LIN {X 0,Y 277.83,Z 467.311,A -85,B 0,C 180,E1 -25540.628,E2 -25540.628} C_VEL
LIN {X 0,Y 277.38,Z 485.512,A -85,B 0,C 180,E1 -25541.504,E2 -25541.504} C_VEL
LIN {X 0,Y 276.723,Z 501.553,A -85,B 0,C 180,E1 -25542.602,E2 -25542.602} C_VEL
LIN {X 0,Y 276.071,Z 515.024,A -85,B 0,C 180,E1 -25543.794,E2 -25543.794} C_VEL
LIN {X 0,Y 275.265,Z 529.451,A -85,B 0,C 180,E1 -25545.393,E2 -25545.393} C_VEL
LIN {X 0,Y 274.573,Z 543.321,A -85,B 0,C 180,E1 -25547.289,E2 -25547.289} C_VEL
LIN {X 0,Y 273.841,Z 555.486,A -85,B 0,C 180,E1 -25549.313,E2 -25549.313} C_VEL
LIN {X 0,Y 273.731,Z 556.96,A -85,B 0,C 180,E1 -25549.589,E2 -25549.589} C_VEL
LIN {X 0,Y 272.791,Z 561.229,A -85,B 0,C 180,E1 -25550.426,E2 -25550.426} C_VEL
LIN {X 0,Y 269.621,Z 567.675,A -85,B 0,C 180,E1 -25551.869,E2 -25551.869} C_VEL
LIN {X 0,Y 266.574,Z 573.805,A -85,B 0,C 180,E1 -25553.418,E2 -25553.418} C_VEL
LIN {X 0,Y 265.838,Z 577.453,A -85,B 0,C 180,E1 -25554.406,E2 -25554.406} C_VEL
LIN {X 0,Y 265.849,Z 586.101,A -85,B 0,C 180,E1 -25556.979,E2 -25556.979} C_VEL
LIN {X 0,Y 266.003,Z 592.424,A -85,B 0,C 180,E1 -25559.245,E2 -25559.245} C_VEL
LIN {X 0,Y 266.684,Z 599.311,A -85,B 0,C 180,E1 -25562.258,E2 -25562.258} C_VEL
LIN {X 0,Y 268.062,Z 604.601,A -85,B 0,C 180,E1 -25565.247,E2 -25565.247} C_VEL
LIN {X 0,Y 269.492,Z 607.656,A -85,B 0,C 180,E1 -25567.467,E2 -25567.467} C_VEL
LIN {X 0,Y 271.89,Z 610.479,A -85,B 0,C 180,E1 -25570.389,E2 -25570.389} C_VEL
LIN {X 0,Y 275.047,Z 611.982,A -85,B 0,C 180,E1 -25573.249,E2 -25573.249} C_VEL
LIN {X 0,Y 276.98,Z 612.223,A -85,B 0,C 180,E1 -25574.648,E2 -25574.648} C_VEL
LIN {X 0,Y 281.552,Z 611.672,A -85,B 0,C 180,E1 -25577.369,E2 -25577.369} C_VEL
LIN {X 0,Y 286.526,Z 609.815,A -85,B 0,C 180,E1 -25580.013,E2 -25580.013} C_VEL
LIN {X 0,Y 292.033,Z 606.641,A -85,B 0,C 180,E1 -25582.567,E2 -25582.567} C_VEL
LIN {X 0,Y 298.202,Z 601.947,A -85,B 0,C 180,E1 -25585.011,E2 -25585.011} C_VEL
LIN {X 0,Y 304.831,Z 595.719,A -85,B 0,C 180,E1 -25587.359,E2 -25587.359} C_VEL
LIN {X 0,Y 310.995,Z 588.827,A -85,B 0,C 180,E1 -25589.332,E2 -25589.332} C_VEL
LIN {X 0,Y 317.678,Z 580.405,A -85,B 0,C 180,E1 -25591.208,E2 -25591.208} C_VEL
LIN {X 0,Y 323.654,Z 571.647,A -85,B 0,C 180,E1 -25592.755,E2 -25592.755} C_VEL
LIN {X 0,Y 329.828,Z 561.351,A -85,B 0,C 180,E1 -25594.247,E2 -25594.247} C_VEL
LIN {X 0,Y 335.133,Z 551.118,A -85,B 0,C 180,E1 -25595.449,E2 -25595.449} C_VEL
LIN {X 0,Y 341.022,Z 537.921,A -85,B 0,C 180,E1 -25596.742,E2 -25596.742} C_VEL
LIN {X 0,Y 345.906,Z 524.621,A -85,B 0,C 180,E1 -25597.774,E2 -25597.774} C_VEL
LIN {X 0,Y 350.516,Z 508.978,A -85,B 0,C 180,E1 -25598.735,E2 -25598.735} C_VEL
LIN {X 0,Y 355.504,Z 486.941,A -85,B 0,C 180,E1 -25599.714,E2 -25599.714} C_VEL
LIN {X 0,Y 359.013,Z 471.3,A -85,B 0,C 180,E1 -25600.286,E2 -25600.286} C_VEL
LIN {X 0,Y 358.746,Z 470.474,A -85,B 0,C 180,E1 -25601.016,E2 -25601.016} C_VEL
LIN {X 0,Y 358.206,Z 469.756,A -85,B 0,C 180,E1 -25603.188,E2 -25603.188} C_VEL
LIN {X 0,Y 358.394,Z 470.084,A -85,B 0,C 180,E1 -25604.963,E2 -25604.963} C_VEL
LIN {X 0,Y 358.539,Z 470.42,A -85,B 0,C 180,E1 -25605.572,E2 -25605.572} C_VEL
LIN {X 0,Y 355.174,Z 487.615,A -85,B 0,C 180,E1 -25607.063,E2 -25607.063} C_VEL
LIN {X 0,Y 352.734,Z 500.618,A -85,B 0,C 180,E1 -25607.993,E2 -25607.993} C_VEL
LIN {X 0,Y 351.508,Z 506.79,A -85,B 0,C 180,E1 -25608.315,E2 -25608.315} C_VEL
LIN {X 0,Y 346.503,Z 527.149,A -85,B 0,C 180,E1 -25609.055,E2 -25609.055} C_VEL
LIN {X 0,Y 340.345,Z 545.929,A -85,B 0,C 180,E1 -25609.897,E2 -25609.897} C_VEL
LIN {X 0,Y 333.914,Z 561.533,A -85,B 0,C 180,E1 -25610.781,E2 -25610.781} C_VEL
LIN {X 0,Y 326.496,Z 576.813,A -85,B 0,C 180,E1 -25611.918,E2 -25611.918} C_VEL
LIN {X 0,Y 319.543,Z 589.349,A -85,B 0,C 180,E1 -25613.125,E2 -25613.125} C_VEL
LIN {X 0,Y 312.972,Z 599.943,A -85,B 0,C 180,E1 -25614.416,E2 -25614.416} C_VEL
LIN {X 0,Y 306.212,Z 609.968,A -85,B 0,C 180,E1 -25615.914,E2 -25615.914} C_VEL
LIN {X 0,Y 298.907,Z 619.806,A -85,B 0,C 180,E1 -25617.784,E2 -25617.784} C_VEL
LIN {X 0,Y 292.343,Z 628.114,A -85,B 0,C 180,E1 -25619.791,E2 -25619.791} C_VEL
LIN {X 0,Y 285.597,Z 635.955,A -85,B 0,C 180,E1 -25622.226,E2 -25622.226} C_VEL
LIN {X 0,Y 279.804,Z 642.289,A -85,B 0,C 180,E1 -25624.813,E2 -25624.813} C_VEL
LIN {X 0,Y 274.862,Z 647.227,A -85,B 0,C 180,E1 -25627.526,E2 -25627.526} C_VEL
LIN {X 0,Y 270.975,Z 650.909,A -85,B 0,C 180,E1 -25630.364,E2 -25630.364} C_VEL
LIN {X 0,Y 268.293,Z 653.413,A -85,B 0,C 180,E1 -25633.31,E2 -25633.31} C_VEL
LIN {X 0,Y 266.458,Z 654.808,A -85,B 0,C 180,E1 -25636.563,E2 -25636.563} C_VEL
LIN {X 0,Y 266.255,Z 655.027,A -85,B 0,C 180,E1 -25637.015,E2 -25637.015} C_VEL
LIN {X 0,Y 265.734,Z 658.417,A -85,B 0,C 180,E1 -25639.367,E2 -25639.367} C_VEL
LIN {X 0,Y 265.875,Z 660.76,A -85,B 0,C 180,E1 -25641.382,E2 -25641.382} C_VEL
LIN {X 0,Y 265.538,Z 670.158,A -85,B 0,C 180,E1 -25643.563,E2 -25643.563} C_VEL
LIN {X 0,Y 265.443,Z 678.349,A -85,B 0,C 180,E1 -25645.838,E2 -25645.838} C_VEL
LIN {X 0,Y 265.218,Z 686.104,A -85,B 0,C 180,E1 -25648.486,E2 -25648.486} C_VEL
LIN {X 0,Y 265.047,Z 691.433,A -85,B 0,C 180,E1 -25650.757,E2 -25650.757} C_VEL
LIN {X 0,Y 264.821,Z 696.988,A -85,B 0,C 180,E1 -25653.791,E2 -25653.791} C_VEL
LIN {X 0,Y 264.9,Z 700.153,A -85,B 0,C 180,E1 -25656.071,E2 -25656.071} C_VEL
LIN {X 0,Y 265.517,Z 703.155,A -85,B 0,C 180,E1 -25659.107,E2 -25659.107} C_VEL
LIN {X 0,Y 267.125,Z 704.904,A -85,B 0,C 180,E1 -25662.109,E2 -25662.109} C_VEL
LIN {X 0,Y 269.559,Z 705.406,A -85,B 0,C 180,E1 -25665.061,E2 -25665.061} C_VEL
LIN {X 0,Y 272.975,Z 704.659,A -85,B 0,C 180,E1 -25667.934,E2 -25667.934} C_VEL
LIN {X 0,Y 276.889,Z 702.698,A -85,B 0,C 180,E1 -25670.742,E2 -25670.742} C_VEL
LIN {X 0,Y 281.856,Z 699.446,A -85,B 0,C 180,E1 -25673.429,E2 -25673.429} C_VEL
LIN {X 0,Y 287.676,Z 694.827,A -85,B 0,C 180,E1 -25675.994,E2 -25675.994} C_VEL
LIN {X 0,Y 294.153,Z 688.78,A -85,B 0,C 180,E1 -25678.44,E2 -25678.44} C_VEL
LIN {X 0,Y 301.384,Z 681.13,A -85,B 0,C 180,E1 -25680.75,E2 -25680.75} C_VEL
LIN {X 0,Y 308.102,Z 673.094,A -85,B 0,C 180,E1 -25682.639,E2 -25682.639} C_VEL
LIN {X 0,Y 315.561,Z 663.159,A -85,B 0,C 180,E1 -25684.473,E2 -25684.473} C_VEL
LIN {X 0,Y 322.247,Z 653.147,A -85,B 0,C 180,E1 -25685.936,E2 -25685.936} C_VEL
LIN {X 0,Y 329.341,Z 641.237,A -85,B 0,C 180,E1 -25687.311,E2 -25687.311} C_VEL
LIN {X 0,Y 336.155,Z 628.196,A -85,B 0,C 180,E1 -25688.499,E2 -25688.499} C_VEL
LIN {X 0,Y 342.004,Z 615.243,A -85,B 0,C 180,E1 -25689.412,E2 -25689.412} C_VEL
LIN {X 0,Y 347.768,Z 600.079,A -85,B 0,C 180,E1 -25690.233,E2 -25690.233} C_VEL
LIN {X 0,Y 352.842,Z 583.368,A -85,B 0,C 180,E1 -25690.927,E2 -25690.927} C_VEL
LIN {X 0,Y 370.753,Z 509.799,A -85,B 0,C 180,E1 -25693.448,E2 -25693.448} C_VEL
LIN {X 0,Y 370.966,Z 508.888,A -85,B 0,C 180,E1 -25693.515,E2 -25693.515} C_VEL
LIN {X 0,Y 370.589,Z 509.38,A -85,B 0,C 180,E1 -25694.543,E2 -25694.543} C_VEL
LIN {X 0,Y 370.186,Z 511.289,A -85,B 0,C 180,E1 -25695.973,E2 -25695.973} C_VEL
LIN {X 0,Y 368.294,Z 519.836,A -85,B 0,C 180,E1 -25696.875,E2 -25696.875} C_VEL
LIN {X 0,Y 352.372,Z 585.479,A -85,B 0,C 180,E1 -25699.122,E2 -25699.122} C_VEL
LIN {X 0,Y 347.28,Z 601.58,A -85,B 0,C 180,E1 -25699.803,E2 -25699.803} C_VEL
LIN {X 0,Y 342.005,Z 615.289,A -85,B 0,C 180,E1 -25700.588,E2 -25700.588} C_VEL
LIN {X 0,Y 335.585,Z 629.314,A -85,B 0,C 180,E1 -25701.615,E2 -25701.615} C_VEL
LIN {X 0,Y 328.309,Z 643.052,A -85,B 0,C 180,E1 -25702.936,E2 -25702.936} C_VEL
LIN {X 0,Y 321.34,Z 654.459,A -85,B 0,C 180,E1 -25704.332,E2 -25704.332} C_VEL
LIN {X 0,Y 313.687,Z 665.565,A -85,B 0,C 180,E1 -25706.066,E2 -25706.066} C_VEL
LIN {X 0,Y 306.92,Z 674.313,A -85,B 0,C 180,E1 -25707.787,E2 -25707.787} C_VEL
LIN {X 0,Y 299.783,Z 682.581,A -85,B 0,C 180,E1 -25709.846,E2 -25709.846} C_VEL
LIN {X 0,Y 292.769,Z 689.758,A -85,B 0,C 180,E1 -25712.191,E2 -25712.191} C_VEL
LIN {X 0,Y 286.491,Z 695.367,A -85,B 0,C 180,E1 -25714.669,E2 -25714.669} C_VEL
LIN {X 0,Y 282.285,Z 698.658,A -85,B 0,C 180,E1 -25716.609,E2 -25716.609} C_VEL
LIN {X 0,Y 277.216,Z 701.896,A -85,B 0,C 180,E1 -25719.284,E2 -25719.284} C_VEL
LIN {X 0,Y 273.238,Z 703.833,A -85,B 0,C 180,E1 -25722.085,E2 -25722.085} C_VEL
LIN {X 0,Y 269.767,Z 704.556,A -85,B 0,C 180,E1 -25724.951,E2 -25724.951} C_VEL
LIN {X 0,Y 267.286,Z 704.033,A -85,B 0,C 180,E1 -25727.899,E2 -25727.899} C_VEL
LIN {X 0,Y 265.594,Z 702.267,A -85,B 0,C 180,E1 -25730.896,E2 -25730.896} C_VEL
LIN {X 0,Y 264.91,Z 699.252,A -85,B 0,C 180,E1 -25733.929,E2 -25733.929} C_VEL
LIN {X 0,Y 264.693,Z 694.866,A -85,B 0,C 180,E1 -25736.967,E2 -25736.967} C_VEL
LIN {X 0,Y 264.902,Z 690.537,A -85,B 0,C 180,E1 -25739.243,E2 -25739.243} C_VEL
LIN {X 0,Y 265.056,Z 685.235,A -85,B 0,C 180,E1 -25741.515,E2 -25741.515} C_VEL
LIN {X 0,Y 265.325,Z 677.568,A -85,B 0,C 180,E1 -25744.164,E2 -25744.164} C_VEL
LIN {X 0,Y 265.522,Z 669.502,A -85,B 0,C 180,E1 -25746.438,E2 -25746.438} C_VEL
LIN {X 0,Y 265.972,Z 659.849,A -85,B 0,C 180,E1 -25748.71,E2 -25748.71} C_VEL
LIN {X 0,Y 266.506,Z 648.108,A -85,B 0,C 180,E1 -25750.985,E2 -25750.985} C_VEL
LIN {X 0,Y 267.25,Z 636.276,A -85,B 0,C 180,E1 -25752.873,E2 -25752.873} C_VEL
LIN {X 0,Y 268.081,Z 622.148,A -85,B 0,C 180,E1 -25754.719,E2 -25754.719} C_VEL
LIN {X 0,Y 268.919,Z 608.368,A -85,B 0,C 180,E1 -25756.164,E2 -25756.164} C_VEL
LIN {X 0,Y 269.645,Z 593.38,A -85,B 0,C 180,E1 -25757.382,E2 -25757.382} C_VEL
LIN {X 0,Y 270.385,Z 577.273,A -85,B 0,C 180,E1 -25758.356,E2 -25758.356} C_VEL
LIN {X 0,Y 274.001,Z 479.005,A -85,B 0,C 180,E1 -25762.85,E2 -25762.85} C_VEL
LIN {X 0,Y 271.934,Z 450.923,A -85,B 0,C 180,E1 -25764.153,E2 -25764.153} C_VEL
LIN {X 0,Y 271.714,Z 439.706,A -85,B 0,C 180,E1 -25764.664,E2 -25764.664} C_VEL
LIN {X 0,Y 274.536,Z 413.307,A -85,B 0,C 180,E1 -25769.311,E2 -25769.311} C_VEL
LIN {X 0,Y 275.637,Z 402.656,A -85,B 0,C 180,E1 -25771.183,E2 -25771.183} C_VEL
LIN {X 0,Y 271.56,Z 383.718,A -85,B 0,C 180,E1 -25774.809,E2 -25774.809} C_VEL
LIN {X 0,Y 267.348,Z 364.742,A -85,B 0,C 180,E1 -25778.599,E2 -25778.599} C_VEL
LIN {X 0,Y 267.282,Z 364.749,A -85,B 0,C 180,E1 -25782.951,E2 -25782.951} C_VEL
LIN {X 0,Y 267.327,Z 364.736,A -85,B 0,C 180,E1 -25785.028,E2 -25785.028} C_VEL
LIN {X 0,Y 267.29,Z 364.739,A -85,B 0,C 180,E1 -25789.461,E2 -25789.461} C_VEL
LIN {X 0,Y 267.315,Z 364.738,A -85,B 0,C 180,E1 -25794.321,E2 -25794.321} C_VEL
LIN {X 0,Y 267.279,Z 364.725,A -85,B 0,C 180,E1 -25798.39,E2 -25798.39} C_VEL
LIN {X 0,Y 267.304,Z 364.747,A -85,B 0,C 180,E1 -25800.955,E2 -25800.955} C_VEL
LIN {X 0,Y 268.431,Z 367.764,A -85,B 0,C 180,E1 -25801.217,E2 -25801.217} C_VEL
LIN {X 0,Y 269.854,Z 370.165,A -85,B 0,C 180,E1 -25801.482,E2 -25801.482} C_VEL
LIN {X 0,Y 277.959,Z 385.073,A -85,B 0,C 180,E1 -25802.963,E2 -25802.963} C_VEL
LIN {X 0,Y 286.368,Z 402.981,A -85,B 0,C 180,E1 -25804.457,E2 -25804.457} C_VEL
LIN {X 0,Y 288.308,Z 407.611,A -85,B 0,C 180,E1 -25804.801,E2 -25804.801} C_VEL
LIN {X 0,Y 286.431,Z 466.207,A -85,B 0,C 180,E1 -25806.228,E2 -25806.228} C_VEL
LIN {X 0,Y 285.998,Z 484.983,A -85,B 0,C 180,E1 -25806.789,E2 -25806.789} C_VEL
LIN {X 0,Y 285.282,Z 499.086,A -85,B 0,C 180,E1 -25807.489,E2 -25807.489} C_VEL
LIN {X 0,Y 284.062,Z 512.189,A -85,B 0,C 180,E1 -25808.387,E2 -25808.387} C_VEL
LIN {X 0,Y 282.505,Z 524.593,A -85,B 0,C 180,E1 -25809.5,E2 -25809.5} C_VEL
LIN {X 0,Y 280.907,Z 536.687,A -85,B 0,C 180,E1 -25810.897,E2 -25810.897} C_VEL
LIN {X 0,Y 278.766,Z 549.061,A -85,B 0,C 180,E1 -25812.659,E2 -25812.659} C_VEL
LIN {X 0,Y 276.419,Z 560.329,A -85,B 0,C 180,E1 -25814.659,E2 -25814.659} C_VEL
LIN {X 0,Y 274.258,Z 569.767,A -85,B 0,C 180,E1 -25816.712,E2 -25816.712} C_VEL
LIN {X 0,Y 272.36,Z 577.943,A -85,B 0,C 180,E1 -25818.879,E2 -25818.879} C_VEL
LIN {X 0,Y 270.78,Z 584.769,A -85,B 0,C 180,E1 -25821.071,E2 -25821.071} C_VEL
LIN {X 0,Y 269.339,Z 590.433,A -85,B 0,C 180,E1 -25823.28,E2 -25823.28} C_VEL
LIN {X 0,Y 268.353,Z 595.066,A -85,B 0,C 180,E1 -25825.509,E2 -25825.509} C_VEL
LIN {X 0,Y 267.32,Z 599.892,A -85,B 0,C 180,E1 -25828.499,E2 -25828.499} C_VEL
LIN {X 0,Y 266.7,Z 603.275,A -85,B 0,C 180,E1 -25831.505,E2 -25831.505} C_VEL
LIN {X 0,Y 266.712,Z 605.29,A -85,B 0,C 180,E1 -25834.519,E2 -25834.519} C_VEL
LIN {X 0,Y 266.94,Z 606.029,A -85,B 0,C 180,E1 -25837.539,E2 -25837.539} C_VEL
LIN {X 0,Y 267.632,Z 605.467,A -85,B 0,C 180,E1 -25840.557,E2 -25840.557} C_VEL
LIN {X 0,Y 268.764,Z 603.589,A -85,B 0,C 180,E1 -25843.566,E2 -25843.566} C_VEL
LIN {X 0,Y 270.604,Z 600.316,A -85,B 0,C 180,E1 -25846.543,E2 -25846.543} C_VEL
LIN {X 0,Y 272.83,Z 595.577,A -85,B 0,C 180,E1 -25849.497,E2 -25849.497} C_VEL
LIN {X 0,Y 275.625,Z 589.204,A -85,B 0,C 180,E1 -25852.408,E2 -25852.408} C_VEL
LIN {X 0,Y 278.481,Z 582.029,A -85,B 0,C 180,E1 -25854.935,E2 -25854.935} C_VEL
LIN {X 0,Y 281.208,Z 574.574,A -85,B 0,C 180,E1 -25857.038,E2 -25857.038} C_VEL
LIN {X 0,Y 284.271,Z 565.532,A -85,B 0,C 180,E1 -25859.12,E2 -25859.12} C_VEL
LIN {X 0,Y 287.348,Z 555.324,A -85,B 0,C 180,E1 -25861.034,E2 -25861.034} C_VEL
LIN {X 0,Y 290.156,Z 544.467,A -85,B 0,C 180,E1 -25862.693,E2 -25862.693} C_VEL
LIN {X 0,Y 292.969,Z 532.202,A -85,B 0,C 180,E1 -25864.184,E2 -25864.184} C_VEL
LIN {X 0,Y 295.052,Z 520.351,A -85,B 0,C 180,E1 -25865.356,E2 -25865.356} C_VEL
LIN {X 0,Y 296.867,Z 506.748,A -85,B 0,C 180,E1 -25866.404,E2 -25866.404} C_VEL
LIN {X 0,Y 298.241,Z 492.635,A -85,B 0,C 180,E1 -25867.193,E2 -25867.193} C_VEL
LIN {X 0,Y 298.945,Z 478.48,A -85,B 0,C 180,E1 -25867.733,E2 -25867.733} C_VEL
LIN {X 0,Y 301.095,Z 422.335,A -85,B 0,C 180,E1 -25869.078,E2 -25869.078} C_VEL
LIN {X 0,Y 291.811,Z 404.264,A -85,B 0,C 180,E1 -25871.027,E2 -25871.027} C_VEL
LIN {X 0,Y 282.758,Z 388.895,A -85,B 0,C 180,E1 -25873.035,E2 -25873.035} C_VEL
LIN {X 0,Y 275.38,Z 377.541,A -85,B 0,C 180,E1 -25874.78,E2 -25874.78} C_VEL
LIN {X 0,Y 272.396,Z 373.287,A -85,B 0,C 180,E1 -25875.515,E2 -25875.515} C_VEL
LIN {X 0,Y 270.318,Z 369.961,A -85,B 0,C 180,E1 -25876.056,E2 -25876.056} C_VEL
LIN {X 0,Y 267.918,Z 367.028,A -85,B 0,C 180,E1 -25876.663,E2 -25876.663} C_VEL
LIN {X 0,Y 267.226,Z 364.754,A -85,B 0,C 180,E1 -25876.91,E2 -25876.91} C_VEL
LIN {X 0,Y 267.229,Z 364.728,A -85,B 0,C 180,E1 -25881.017,E2 -25881.017} C_VEL
LIN {X 0,Y 267.291,Z 364.703,A -85,B 0,C 180,E1 -25884.793,E2 -25884.793} C_VEL
LIN {X 0,Y 267.263,Z 364.739,A -85,B 0,C 180,E1 -25888.388,E2 -25888.388} C_VEL
LIN {X 0,Y 267.297,Z 364.747,A -85,B 0,C 180,E1 -25891.856,E2 -25891.856} C_VEL
LIN {X 0,Y 267.426,Z 364.728,A -85,B 0,C 180,E1 -25895.99,E2 -25895.99} C_VEL
LIN {X 0,Y 272.348,Z 385.825,A -85,B 0,C 180,E1 -25897.034,E2 -25897.034} C_VEL
LIN {X 0,Y 273.158,Z 389.512,A -85,B 0,C 180,E1 -25897.208,E2 -25897.208} C_VEL
LIN {X 0,Y 270.75,Z 467.378,A -85,B 0,C 180,E1 -25900.642,E2 -25900.642} C_VEL
LIN {X 0,Y 270.245,Z 486.31,A -85,B 0,C 180,E1 -25901.585,E2 -25901.585} C_VEL
LIN {X 0,Y 269.623,Z 502.271,A -85,B 0,C 180,E1 -25902.714,E2 -25902.714} C_VEL
LIN {X 0,Y 268.919,Z 515.677,A -85,B 0,C 180,E1 -25903.933,E2 -25903.933} C_VEL
LIN {X 0,Y 268.125,Z 529.839,A -85,B 0,C 180,E1 -25905.535,E2 -25905.535} C_VEL
LIN {X 0,Y 267.496,Z 542.755,A -85,B 0,C 180,E1 -25907.332,E2 -25907.332} C_VEL
LIN {X 0,Y 266.77,Z 555.138,A -85,B 0,C 180,E1 -25909.409,E2 -25909.409} C_VEL
LIN {X 0,Y 266.187,Z 566.344,A -85,B 0,C 180,E1 -25911.678,E2 -25911.678} C_VEL
LIN {X 0,Y 265.879,Z 575.75,A -85,B 0,C 180,E1 -25913.951,E2 -25913.951} C_VEL
LIN {X 0,Y 265.838,Z 577.453,A -85,B 0,C 180,E1 -25914.406,E2 -25914.406} C_VEL
LIN {X 0,Y 265.112,Z 581.008,A -85,B 0,C 180,E1 -25915.414,E2 -25915.414} C_VEL
LIN {X 0,Y 262.22,Z 586.278,A -85,B 0,C 180,E1 -25917.134,E2 -25917.134} C_VEL
LIN {X 0,Y 259.493,Z 591.072,A -85,B 0,C 180,E1 -25918.959,E2 -25918.959} C_VEL
LIN {X 0,Y 259.039,Z 593.889,A -85,B 0,C 180,E1 -25920.111,E2 -25920.111} C_VEL
LIN {X 0,Y 259.883,Z 600.448,A -85,B 0,C 180,E1 -25923.09,E2 -25923.09} C_VEL
LIN {X 0,Y 261.463,Z 605.721,A -85,B 0,C 180,E1 -25926.151,E2 -25926.151} C_VEL
LIN {X 0,Y 263.606,Z 609.564,A -85,B 0,C 180,E1 -25929.173,E2 -25929.173} C_VEL
LIN {X 0,Y 266.45,Z 612.093,A -85,B 0,C 180,E1 -25932.14,E2 -25932.14} C_VEL
LIN {X 0,Y 270.194,Z 613.285,A -85,B 0,C 180,E1 -25935.024,E2 -25935.024} C_VEL
LIN {X 0,Y 274.934,Z 613.1,A -85,B 0,C 180,E1 -25937.801,E2 -25937.801} C_VEL
LIN {X 0,Y 280.088,Z 611.623,A -85,B 0,C 180,E1 -25940.494,E2 -25940.494} C_VEL
LIN {X 0,Y 285.763,Z 608.805,A -85,B 0,C 180,E1 -25943.09,E2 -25943.09} C_VEL
LIN {X 0,Y 292.141,Z 604.553,A -85,B 0,C 180,E1 -25945.567,E2 -25945.567} C_VEL
LIN {X 0,Y 299.02,Z 598.792,A -85,B 0,C 180,E1 -25947.936,E2 -25947.936} C_VEL
LIN {X 0,Y 304.456,Z 593.433,A -85,B 0,C 180,E1 -25949.646,E2 -25949.646} C_VEL
LIN {X 0,Y 311.254,Z 585.766,A -85,B 0,C 180,E1 -25951.548,E2 -25951.548} C_VEL
LIN {X 0,Y 318.426,Z 576.444,A -85,B 0,C 180,E1 -25953.362,E2 -25953.362} C_VEL
LIN {X 0,Y 324.796,Z 566.796,A -85,B 0,C 180,E1 -25954.854,E2 -25954.854} C_VEL
LIN {X 0,Y 331.368,Z 555.391,A -85,B 0,C 180,E1 -25956.289,E2 -25956.289} C_VEL
LIN {X 0,Y 337.49,Z 542.805,A -85,B 0,C 180,E1 -25957.565,E2 -25957.565} C_VEL
LIN {X 0,Y 343.133,Z 528.947,A -85,B 0,C 180,E1 -25958.693,E2 -25958.693} C_VEL
LIN {X 0,Y 347.531,Z 515.703,A -85,B 0,C 180,E1 -25959.551,E2 -25959.551} C_VEL
LIN {X 0,Y 351.216,Z 501.453,A -85,B 0,C 180,E1 -25960.267,E2 -25960.267} C_VEL
LIN {X 0,Y 356.888,Z 477.219,A -85,B 0,C 180,E1 -25961.231,E2 -25961.231} C_VEL
LIN {X 0,Y 356.421,Z 476.612,A -85,B 0,C 180,E1 -25963.458,E2 -25963.458} C_VEL
LIN {X 0,Y 356.573,Z 477.056,A -85,B 0,C 180,E1 -25964.894,E2 -25964.894} C_VEL
LIN {X 0,Y 352.97,Z 493.856,A -85,B 0,C 180,E1 -25966.302,E2 -25966.302} C_VEL
LIN {X 0,Y 350.92,Z 503.807,A -85,B 0,C 180,E1 -25966.985,E2 -25966.985} C_VEL
LIN {X 0,Y 349.828,Z 508.728,A -85,B 0,C 180,E1 -25967.223,E2 -25967.223} C_VEL
LIN {X 0,Y 344.858,Z 527.571,A -85,B 0,C 180,E1 -25967.912,E2 -25967.912} C_VEL
LIN {X 0,Y 339.896,Z 542.17,A -85,B 0,C 180,E1 -25968.546,E2 -25968.546} C_VEL
LIN {X 0,Y 333.423,Z 557.718,A -85,B 0,C 180,E1 -25969.365,E2 -25969.365} C_VEL
LIN {X 0,Y 326.491,Z 571.926,A -85,B 0,C 180,E1 -25970.338,E2 -25970.338} C_VEL
LIN {X 0,Y 319.15,Z 584.979,A -85,B 0,C 180,E1 -25971.482,E2 -25971.482} C_VEL
LIN {X 0,Y 310.953,Z 597.878,A -85,B 0,C 180,E1 -25972.946,E2 -25972.946} C_VEL
LIN {X 0,Y 302.744,Z 609.408,A -85,B 0,C 180,E1 -25974.661,E2 -25974.661} C_VEL
LIN {X 0,Y 295.073,Z 619.163,A -85,B 0,C 180,E1 -25976.502,E2 -25976.502} C_VEL
LIN {X 0,Y 288.155,Z 627.279,A -85,B 0,C 180,E1 -25978.491,E2 -25978.491} C_VEL
LIN {X 0,Y 281.031,Z 635.035,A -85,B 0,C 180,E1 -25980.92,E2 -25980.92} C_VEL
LIN {X 0,Y 274.841,Z 641.231,A -85,B 0,C 180,E1 -25983.513,E2 -25983.513} C_VEL
LIN {X 0,Y 269.486,Z 646.112,A -85,B 0,C 180,E1 -25986.242,E2 -25986.242} C_VEL
LIN {X 0,Y 266.188,Z 648.922,A -85,B 0,C 180,E1 -25988.383,E2 -25988.383} C_VEL
LIN {X 0,Y 262.769,Z 651.676,A -85,B 0,C 180,E1 -25991.344,E2 -25991.344} C_VEL
LIN {X 0,Y 260.453,Z 653.292,A -85,B 0,C 180,E1 -25994.399,E2 -25994.399} C_VEL
LIN {X 0,Y 259.495,Z 653.822,A -85,B 0,C 180,E1 -25996.344,E2 -25996.344} C_VEL
LIN {X 0,Y 258.674,Z 657.708,A -85,B 0,C 180,E1 -25999.073,E2 -25999.073} C_VEL
LIN {X 0,Y 258.897,Z 660.585,A -85,B 0,C 180,E1 -26001.736,E2 -26001.736} C_VEL
LIN {X 0,Y 258.58,Z 670.73,A -85,B 0,C 180,E1 -26004.17,E2 -26004.17} C_VEL
LIN {X 0,Y 258.424,Z 678.75,A -85,B 0,C 180,E1 -26006.503,E2 -26006.503} C_VEL
LIN {X 0,Y 258.242,Z 686.361,A -85,B 0,C 180,E1 -26009.223,E2 -26009.223} C_VEL
LIN {X 0,Y 257.992,Z 691.58,A -85,B 0,C 180,E1 -26011.556,E2 -26011.556} C_VEL
LIN {X 0,Y 257.827,Z 697.043,A -85,B 0,C 180,E1 -26014.675,E2 -26014.675} C_VEL
LIN {X 0,Y 258.192,Z 701.017,A -85,B 0,C 180,E1 -26017.796,E2 -26017.796} C_VEL
LIN {X 0,Y 259.311,Z 703.677,A -85,B 0,C 180,E1 -26020.899,E2 -26020.899} C_VEL
LIN {X 0,Y 261.278,Z 705.098,A -85,B 0,C 180,E1 -26023.962,E2 -26023.962} C_VEL
LIN {X 0,Y 264.39,Z 705.301,A -85,B 0,C 180,E1 -26026.943,E2 -26026.943} C_VEL
LIN {X 0,Y 268.81,Z 704.046,A -85,B 0,C 180,E1 -26030.273,E2 -26030.273} C_VEL
LIN {X 0,Y 272.73,Z 702.051,A -85,B 0,C 180,E1 -26032.659,E2 -26032.659} C_VEL
LIN {X 0,Y 278.344,Z 698.529,A -85,B 0,C 180,E1 -26035.328,E2 -26035.328} C_VEL
LIN {X 0,Y 284.711,Z 693.66,A -85,B 0,C 180,E1 -26037.868,E2 -26037.868} C_VEL
LIN {X 0,Y 291.728,Z 687.369,A -85,B 0,C 180,E1 -26040.279,E2 -26040.279} C_VEL
LIN {X 0,Y 299.519,Z 679.422,A -85,B 0,C 180,E1 -26042.539,E2 -26042.539} C_VEL
LIN {X 0,Y 306.796,Z 671.005,A -85,B 0,C 180,E1 -26044.384,E2 -26044.384} C_VEL
LIN {X 0,Y 314.634,Z 660.781,A -85,B 0,C 180,E1 -26046.153,E2 -26046.153} C_VEL
LIN {X 0,Y 321.729,Z 650.406,A -85,B 0,C 180,E1 -26047.56,E2 -26047.56} C_VEL
LIN {X 0,Y 329.209,Z 638.069,A -85,B 0,C 180,E1 -26048.878,E2 -26048.878} C_VEL
LIN {X 0,Y 335.705,Z 625.761,A -85,B 0,C 180,E1 -26049.911,E2 -26049.911} C_VEL
LIN {X 0,Y 341.79,Z 612.393,A -85,B 0,C 180,E1 -26050.785,E2 -26050.785} C_VEL
LIN {X 0,Y 347.091,Z 598.663,A -85,B 0,C 180,E1 -26051.468,E2 -26051.468} C_VEL
LIN {X 0,Y 352.232,Z 581.967,A -85,B 0,C 180,E1 -26052.132,E2 -26052.132} C_VEL
LIN {X 0,Y 368.84,Z 516.135,A -85,B 0,C 180,E1 -26054.345,E2 -26054.345} C_VEL
LIN {X 0,Y 368.451,Z 517.506,A -85,B 0,C 180,E1 -26055.333,E2 -26055.333} C_VEL
LIN {X 0,Y 367.139,Z 522.804,A -85,B 0,C 180,E1 -26055.858,E2 -26055.858} C_VEL
LIN {X 0,Y 351.021,Z 586.537,A -85,B 0,C 180,E1 -26058.003,E2 -26058.003} C_VEL
LIN {X 0,Y 345.721,Z 602.529,A -85,B 0,C 180,E1 -26058.668,E2 -26058.668} C_VEL
LIN {X 0,Y 340.45,Z 615.613,A -85,B 0,C 180,E1 -26059.409,E2 -26059.409} C_VEL
LIN {X 0,Y 333.766,Z 629.565,A -85,B 0,C 180,E1 -26060.398,E2 -26060.398} C_VEL
LIN {X 0,Y 326.204,Z 643.2,A -85,B 0,C 180,E1 -26061.683,E2 -26061.683} C_VEL
LIN {X 0,Y 318.346,Z 655.386,A -85,B 0,C 180,E1 -26063.161,E2 -26063.161} C_VEL
LIN {X 0,Y 310.363,Z 666.314,A -85,B 0,C 180,E1 -26064.866,E2 -26064.866} C_VEL
LIN {X 0,Y 302.723,Z 675.589,A -85,B 0,C 180,E1 -26066.719,E2 -26066.719} C_VEL
LIN {X 0,Y 295.835,Z 683.014,A -85,B 0,C 180,E1 -26068.608,E2 -26068.608} C_VEL
LIN {X 0,Y 288.431,Z 690.055,A -85,B 0,C 180,E1 -26070.942,E2 -26070.942} C_VEL
LIN {X 0,Y 281.762,Z 695.579,A -85,B 0,C 180,E1 -26073.419,E2 -26073.419} C_VEL
LIN {X 0,Y 275.872,Z 699.716,A -85,B 0,C 180,E1 -26076.031,E2 -26076.031} C_VEL
LIN {X 0,Y 270.638,Z 702.571,A -85,B 0,C 180,E1 -26078.757,E2 -26078.757} C_VEL
LIN {X 0,Y 266.498,Z 704.164,A -85,B 0,C 180,E1 -26081.615,E2 -26081.615} C_VEL
LIN {X 0,Y 262.929,Z 704.554,A -85,B 0,C 180,E1 -26084.55,E2 -26084.55} C_VEL
LIN {X 0,Y 260.363,Z 703.721,A -85,B 0,C 180,E1 -26087.572,E2 -26087.572} C_VEL
LIN {X 0,Y 258.605,Z 701.653,A -85,B 0,C 180,E1 -26090.648,E2 -26090.648} C_VEL
LIN {X 0,Y 257.922,Z 698.341,A -85,B 0,C 180,E1 -26093.764,E2 -26093.764} C_VEL
LIN {X 0,Y 257.722,Z 693.634,A -85,B 0,C 180,E1 -26096.884,E2 -26096.884} C_VEL
LIN {X 0,Y 257.927,Z 689.132,A -85,B 0,C 180,E1 -26099.222,E2 -26099.222} C_VEL
LIN {X 0,Y 258.151,Z 682.505,A -85,B 0,C 180,E1 -26101.944,E2 -26101.944} C_VEL
LIN {X 0,Y 258.382,Z 675.549,A -85,B 0,C 180,E1 -26104.276,E2 -26104.276} C_VEL
LIN {X 0,Y 258.601,Z 667.117,A -85,B 0,C 180,E1 -26106.611,E2 -26106.611} C_VEL
LIN {X 0,Y 259.077,Z 656.97,A -85,B 0,C 180,E1 -26108.944,E2 -26108.944} C_VEL
LIN {X 0,Y 259.668,Z 644.641,A -85,B 0,C 180,E1 -26111.278,E2 -26111.278} C_VEL
LIN {X 0,Y 260.321,Z 633.523,A -85,B 0,C 180,E1 -26113.024,E2 -26113.024} C_VEL
LIN {X 0,Y 261.125,Z 619.696,A -85,B 0,C 180,E1 -26114.808,E2 -26114.808} C_VEL
LIN {X 0,Y 262.021,Z 605.172,A -85,B 0,C 180,E1 -26116.302,E2 -26116.302} C_VEL
LIN {X 0,Y 262.794,Z 589.481,A -85,B 0,C 180,E1 -26117.549,E2 -26117.549} C_VEL
LIN {X 0,Y 263.494,Z 571.773,A -85,B 0,C 180,E1 -26118.552,E2 -26118.552} C_VEL
LIN {X 0,Y 266.897,Z 479.035,A -85,B 0,C 180,E1 -26122.94,E2 -26122.94} C_VEL
LIN {X 0,Y 264.859,Z 450.916,A -85,B 0,C 180,E1 -26124.278,E2 -26124.278} C_VEL
LIN {X 0,Y 264.654,Z 439.51,A -85,B 0,C 180,E1 -26124.845,E2 -26124.845} C_VEL
LIN {X 0,Y 267.455,Z 414.119,A -85,B 0,C 180,E1 -26129.41,E2 -26129.41} C_VEL
LIN {X 0,Y 268.58,Z 404.657,A -85,B 0,C 180,E1 -26131.102,E2 -26131.102} C_VEL
LIN {X 0,Y 267.927,Z 400.271,A -85,B 0,C 180,E1 -26131.936,E2 -26131.936} C_VEL
LIN {X 0,Y 262.929,Z 377.417,A -85,B 0,C 180,E1 -26136.442,E2 -26136.442} C_VEL
LIN {X 0,Y 260.29,Z 365.621,A -85,B 0,C 180,E1 -26138.883,E2 -26138.883} C_VEL
LIN {X 0,Y 260.224,Z 365.628,A -85,B 0,C 180,E1 -26143.385,E2 -26143.385} C_VEL
LIN {X 0,Y 260.224,Z 365.623,A -85,B 0,C 180,E1 -26146.616,E2 -26146.616} C_VEL
LIN {X 0,Y 260.247,Z 365.615,A -85,B 0,C 180,E1 -26149.763,E2 -26149.763} C_VEL
LIN {X 0,Y 260.235,Z 365.618,A -85,B 0,C 180,E1 -26153.851,E2 -26153.851} C_VEL
LIN {X 0,Y 260.236,Z 365.604,A -85,B 0,C 180,E1 -26157.431,E2 -26157.431} C_VEL
LIN {X 0,Y 260.274,Z 365.61,A -85,B 0,C 180,E1 -26159.975,E2 -26159.975} C_VEL
LIN {X 0,Y 261.23,Z 368.38,A -85,B 0,C 180,E1 -26160.232,E2 -26160.232} C_VEL
LIN {X 0,Y 262.771,Z 370.939,A -85,B 0,C 180,E1 -26160.535,E2 -26160.535} C_VEL
LIN {X 0,Y 271.145,Z 386.061,A -85,B 0,C 180,E1 -26162.138,E2 -26162.138} C_VEL
LIN {X 0,Y 278.882,Z 402.132,A -85,B 0,C 180,E1 -26163.573,E2 -26163.573} C_VEL
LIN {X 0,Y 282.103,Z 409.831,A -85,B 0,C 180,E1 -26164.17,E2 -26164.17} C_VEL
LIN {X 0,Y 280.216,Z 463.43,A -85,B 0,C 180,E1 -26165.491,E2 -26165.491} C_VEL
LIN {X 0,Y 279.698,Z 484.841,A -85,B 0,C 180,E1 -26166.117,E2 -26166.117} C_VEL
LIN {X 0,Y 278.947,Z 499.533,A -85,B 0,C 180,E1 -26166.851,E2 -26166.851} C_VEL
LIN {X 0,Y 277.689,Z 512.717,A -85,B 0,C 180,E1 -26167.768,E2 -26167.768} C_VEL
LIN {X 0,Y 275.972,Z 526.036,A -85,B 0,C 180,E1 -26168.992,E2 -26168.992} C_VEL
LIN {X 0,Y 274.298,Z 538.003,A -85,B 0,C 180,E1 -26170.418,E2 -26170.418} C_VEL
LIN {X 0,Y 272.313,Z 549.027,A -85,B 0,C 180,E1 -26172.021,E2 -26172.021} C_VEL
LIN {X 0,Y 269.933,Z 560.283,A -85,B 0,C 180,E1 -26174.026,E2 -26174.026} C_VEL
LIN {X 0,Y 267.427,Z 570.819,A -85,B 0,C 180,E1 -26176.366,E2 -26176.366} C_VEL
LIN {X 0,Y 265.189,Z 580.152,A -85,B 0,C 180,E1 -26178.96,E2 -26178.96} C_VEL
LIN {X 0,Y 263.264,Z 587.719,A -85,B 0,C 180,E1 -26181.586,E2 -26181.586} C_VEL
LIN {X 0,Y 262.012,Z 592.991,A -85,B 0,C 180,E1 -26183.862,E2 -26183.862} C_VEL
LIN {X 0,Y 260.761,Z 598.553,A -85,B 0,C 180,E1 -26186.921,E2 -26186.921} C_VEL
LIN {X 0,Y 259.859,Z 602.615,A -85,B 0,C 180,E1 -26190,E2 -26190} C_VEL
LIN {X 0,Y 259.593,Z 605.269,A -85,B 0,C 180,E1 -26193.094,E2 -26193.094} C_VEL
LIN {X 0,Y 259.725,Z 606.611,A -85,B 0,C 180,E1 -26196.193,E2 -26196.193} C_VEL
LIN {X 0,Y 260.236,Z 606.662,A -85,B 0,C 180,E1 -26199.294,E2 -26199.294} C_VEL
LIN {X 0,Y 261.168,Z 605.415,A -85,B 0,C 180,E1 -26202.39,E2 -26202.39} C_VEL
LIN {X 0,Y 262.812,Z 602.809,A -85,B 0,C 180,E1 -26205.458,E2 -26205.458} C_VEL
LIN {X 0,Y 264.912,Z 598.789,A -85,B 0,C 180,E1 -26208.499,E2 -26208.499} C_VEL
LIN {X 0,Y 267.54,Z 593.219,A -85,B 0,C 180,E1 -26211.502,E2 -26211.502} C_VEL
LIN {X 0,Y 269.855,Z 587.895,A -85,B 0,C 180,E1 -26213.724,E2 -26213.724} C_VEL
LIN {X 0,Y 272.921,Z 580.244,A -85,B 0,C 180,E1 -26216.278,E2 -26216.278} C_VEL
LIN {X 0,Y 275.914,Z 572.215,A -85,B 0,C 180,E1 -26218.424,E2 -26218.424} C_VEL
LIN {X 0,Y 279.26,Z 562.499,A -85,B 0,C 180,E1 -26220.525,E2 -26220.525} C_VEL
LIN {X 0,Y 282.28,Z 551.868,A -85,B 0,C 180,E1 -26222.415,E2 -26222.415} C_VEL
LIN {X 0,Y 285.488,Z 539.598,A -85,B 0,C 180,E1 -26224.142,E2 -26224.142} C_VEL
LIN {X 0,Y 288.103,Z 527.58,A -85,B 0,C 180,E1 -26225.483,E2 -26225.483} C_VEL
LIN {X 0,Y 290.19,Z 514.189,A -85,B 0,C 180,E1 -26226.685,E2 -26226.685} C_VEL
LIN {X 0,Y 291.804,Z 500.393,A -85,B 0,C 180,E1 -26227.614,E2 -26227.614} C_VEL
LIN {X 0,Y 292.934,Z 485.686,A -85,B 0,C 180,E1 -26228.305,E2 -26228.305} C_VEL
LIN {X 0,Y 293.617,Z 466.227,A -85,B 0,C 180,E1 -26228.863,E2 -26228.863} C_VEL
LIN {X 0,Y 295.369,Z 424.758,A -85,B 0,C 180,E1 -26229.849,E2 -26229.849} C_VEL
LIN {X 0,Y 286.57,Z 407.52,A -85,B 0,C 180,E1 -26231.777,E2 -26231.777} C_VEL
LIN {X 0,Y 277.8,Z 392.689,A -85,B 0,C 180,E1 -26233.802,E2 -26233.802} C_VEL
LIN {X 0,Y 271.267,Z 382.551,A -85,B 0,C 180,E1 -26235.41,E2 -26235.41} C_VEL
LIN {X 0,Y 265.591,Z 374.34,A -85,B 0,C 180,E1 -26236.887,E2 -26236.887} C_VEL
LIN {X 0,Y 263.527,Z 371.229,A -85,B 0,C 180,E1 -26237.455,E2 -26237.455} C_VEL
LIN {X 0,Y 262.754,Z 370.256,A -85,B 0,C 180,E1 -26237.664,E2 -26237.664} C_VEL
LIN {X 0,Y 260.878,Z 367.987,A -85,B 0,C 180,E1 -26238.176,E2 -26238.176} C_VEL
LIN {X 0,Y 260.156,Z 365.629,A -85,B 0,C 180,E1 -26238.458,E2 -26238.458} C_VEL
LIN {X 0,Y 260.184,Z 365.59,A -85,B 0,C 180,E1 -26241.743,E2 -26241.743} C_VEL
LIN {X 0,Y 260.224,Z 365.597,A -85,B 0,C 180,E1 -26245.579,E2 -26245.579} C_VEL
LIN {X 0,Y 260.201,Z 365.613,A -85,B 0,C 180,E1 -26249.477,E2 -26249.477} C_VEL
LIN {X 0,Y 260.271,Z 365.614,A -85,B 0,C 180,E1 -26252.773,E2 -26252.773} C_VEL
LIN {X 0,Y 260.402,Z 365.698,A -85,B 0,C 180,E1 -26255.925,E2 -26255.925} C_VEL
LIN {X 0,Y 265.125,Z 386.28,A -85,B 0,C 180,E1 -26256.947,E2 -26256.947} C_VEL
LIN {X 0,Y 266.034,Z 390.466,A -85,B 0,C 180,E1 -26257.15,E2 -26257.15} C_VEL
LIN {X 0,Y 263.684,Z 465.922,A -85,B 0,C 180,E1 -26260.606,E2 -26260.606} C_VEL
LIN {X 0,Y 263.154,Z 486.103,A -85,B 0,C 180,E1 -26261.624,E2 -26261.624} C_VEL
LIN {X 0,Y 262.567,Z 501.736,A -85,B 0,C 180,E1 -26262.735,E2 -26262.735} C_VEL
LIN {X 0,Y 261.79,Z 516.227,A -85,B 0,C 180,E1 -26264.082,E2 -26264.082} C_VEL
LIN {X 0,Y 261.013,Z 530.486,A -85,B 0,C 180,E1 -26265.741,E2 -26265.741} C_VEL
LIN {X 0,Y 260.346,Z 543.31,A -85,B 0,C 180,E1 -26267.57,E2 -26267.57} C_VEL
LIN {X 0,Y 259.63,Z 555.725,A -85,B 0,C 180,E1 -26269.704,E2 -26269.704} C_VEL
LIN {X 0,Y 259.036,Z 567.778,A -85,B 0,C 180,E1 -26272.229,E2 -26272.229} C_VEL
LIN {X 0,Y 258.781,Z 577.099,A -85,B 0,C 180,E1 -26274.564,E2 -26274.564} C_VEL
LIN {X 0,Y 258.789,Z 586.162,A -85,B 0,C 180,E1 -26277.285,E2 -26277.285} C_VEL
LIN {X 0,Y 259.039,Z 593.889,A -85,B 0,C 180,E1 -26280.111,E2 -26280.111} C_VEL
LIN {X 0,Y 258.671,Z 596.575,A -85,B 0,C 180,E1 -26281.272,E2 -26281.272} C_VEL
LIN {X 0,Y 256.458,Z 600.553,A -85,B 0,C 180,E1 -26283.232,E2 -26283.232} C_VEL
LIN {X 0,Y 254.502,Z 604.039,A -85,B 0,C 180,E1 -26285.272,E2 -26285.272} C_VEL
LIN {X 0,Y 254.547,Z 605.958,A -85,B 0,C 180,E1 -26286.533,E2 -26286.533} C_VEL
LIN {X 0,Y 256.628,Z 609.854,A -85,B 0,C 180,E1 -26289.425,E2 -26289.425} C_VEL
LIN {X 0,Y 259.539,Z 612.698,A -85,B 0,C 180,E1 -26292.468,E2 -26292.468} C_VEL
LIN {X 0,Y 263.421,Z 614.225,A -85,B 0,C 180,E1 -26295.42,E2 -26295.42} C_VEL
LIN {X 0,Y 268.296,Z 614.397,A -85,B 0,C 180,E1 -26298.257,E2 -26298.257} C_VEL
LIN {X 0,Y 273.63,Z 613.293,A -85,B 0,C 180,E1 -26301,E2 -26301} C_VEL
LIN {X 0,Y 279.521,Z 610.893,A -85,B 0,C 180,E1 -26303.637,E2 -26303.637} C_VEL
LIN {X 0,Y 286.095,Z 607.103,A -85,B 0,C 180,E1 -26306.148,E2 -26306.148} C_VEL
LIN {X 0,Y 293.206,Z 601.842,A -85,B 0,C 180,E1 -26308.54,E2 -26308.54} C_VEL
LIN {X 0,Y 300.77,Z 594.957,A -85,B 0,C 180,E1 -26310.82,E2 -26310.82} C_VEL
LIN {X 0,Y 308.942,Z 586.267,A -85,B 0,C 180,E1 -26312.965,E2 -26312.965} C_VEL
LIN {X 0,Y 316.467,Z 576.719,A -85,B 0,C 180,E1 -26314.745,E2 -26314.745} C_VEL
LIN {X 0,Y 323.145,Z 567.072,A -85,B 0,C 180,E1 -26316.204,E2 -26316.204} C_VEL
LIN {X 0,Y 329.725,Z 555.97,A -85,B 0,C 180,E1 -26317.547,E2 -26317.547} C_VEL
LIN {X 0,Y 335.803,Z 544.098,A -85,B 0,C 180,E1 -26318.738,E2 -26318.738} C_VEL
LIN {X 0,Y 341.645,Z 530.28,A -85,B 0,C 180,E1 -26319.843,E2 -26319.843} C_VEL
LIN {X 0,Y 346.375,Z 516.714,A -85,B 0,C 180,E1 -26320.706,E2 -26320.706} C_VEL
LIN {X 0,Y 350.277,Z 502.461,A -85,B 0,C 180,E1 -26321.406,E2 -26321.406} C_VEL
LIN {X 0,Y 354.774,Z 483.686,A -85,B 0,C 180,E1 -26322.165,E2 -26322.165} C_VEL
LIN {X 0,Y 354.688,Z 483.533,A -85,B 0,C 180,E1 -26324.167,E2 -26324.167} C_VEL
LIN {X 0,Y 351.52,Z 497.232,A -85,B 0,C 180,E1 -26325.304,E2 -26325.304} C_VEL
LIN {X 0,Y 349.393,Z 506.697,A -85,B 0,C 180,E1 -26325.947,E2 -26325.947} C_VEL
LIN {X 0,Y 346.864,Z 516.8,A -85,B 0,C 180,E1 -26326.333,E2 -26326.333} C_VEL
LIN {X 0,Y 341.777,Z 533.044,A -85,B 0,C 180,E1 -26326.944,E2 -26326.944} C_VEL
LIN {X 0,Y 334.839,Z 550.633,A -85,B 0,C 180,E1 -26327.777,E2 -26327.777} C_VEL
LIN {X 0,Y 328.26,Z 564.446,A -85,B 0,C 180,E1 -26328.587,E2 -26328.587} C_VEL
LIN {X 0,Y 320.494,Z 578.438,A -85,B 0,C 180,E1 -26329.649,E2 -26329.649} C_VEL
LIN {X 0,Y 313.146,Z 590.243,A -85,B 0,C 180,E1 -26330.809,E2 -26330.809} C_VEL
LIN {X 0,Y 305.488,Z 601.119,A -85,B 0,C 180,E1 -26332.168,E2 -26332.168} C_VEL
LIN {X 0,Y 297.093,Z 611.911,A -85,B 0,C 180,E1 -26333.884,E2 -26333.884} C_VEL
LIN {X 0,Y 289.278,Z 620.951,A -85,B 0,C 180,E1 -26335.738,E2 -26335.738} C_VEL
LIN {X 0,Y 282.214,Z 628.581,A -85,B 0,C 180,E1 -26337.749,E2 -26337.749} C_VEL
LIN {X 0,Y 274.894,Z 635.769,A -85,B 0,C 180,E1 -26340.206,E2 -26340.206} C_VEL
LIN {X 0,Y 268.529,Z 641.549,A -85,B 0,C 180,E1 -26342.84,E2 -26342.84} C_VEL
LIN {X 0,Y 264.304,Z 645.018,A -85,B 0,C 180,E1 -26344.911,E2 -26344.911} C_VEL
LIN {X 0,Y 259.6,Z 648.596,A -85,B 0,C 180,E1 -26347.806,E2 -26347.806} C_VEL
LIN {X 0,Y 256.018,Z 651.024,A -85,B 0,C 180,E1 -26350.833,E2 -26350.833} C_VEL
LIN {X 0,Y 253.632,Z 652.337,A -85,B 0,C 180,E1 -26353.968,E2 -26353.968} C_VEL
LIN {X 0,Y 252.726,Z 652.708,A -85,B 0,C 180,E1 -26355.692,E2 -26355.692} C_VEL
LIN {X 0,Y 251.617,Z 656.999,A -85,B 0,C 180,E1 -26358.763,E2 -26358.763} C_VEL
LIN {X 0,Y 251.887,Z 660.341,A -85,B 0,C 180,E1 -26362.108,E2 -26362.108} C_VEL
LIN {X 0,Y 251.599,Z 671.188,A -85,B 0,C 180,E1 -26364.809,E2 -26364.809} C_VEL
LIN {X 0,Y 251.45,Z 679.088,A -85,B 0,C 180,E1 -26367.206,E2 -26367.206} C_VEL
LIN {X 0,Y 251.27,Z 686.554,A -85,B 0,C 180,E1 -26370,E2 -26370} C_VEL
LIN {X 0,Y 250.954,Z 691.669,A -85,B 0,C 180,E1 -26372.399,E2 -26372.399} C_VEL
LIN {X 0,Y 250.849,Z 695.859,A -85,B 0,C 180,E1 -26374.805,E2 -26374.805} C_VEL
LIN {X 0,Y 251.198,Z 700.13,A -85,B 0,C 180,E1 -26378.014,E2 -26378.014} C_VEL
LIN {X 0,Y 252.37,Z 703.096,A -85,B 0,C 180,E1 -26381.203,E2 -26381.203} C_VEL
LIN {X 0,Y 254.401,Z 704.83,A -85,B 0,C 180,E1 -26384.347,E2 -26384.347} C_VEL
LIN {X 0,Y 257.601,Z 705.37,A -85,B 0,C 180,E1 -26387.403,E2 -26387.403} C_VEL
LIN {X 0,Y 261.766,Z 704.625,A -85,B 0,C 180,E1 -26390.522,E2 -26390.522} C_VEL
LIN {X 0,Y 266.239,Z 702.837,A -85,B 0,C 180,E1 -26393.243,E2 -26393.243} C_VEL
LIN {X 0,Y 272.041,Z 699.712,A -85,B 0,C 180,E1 -26395.958,E2 -26395.958} C_VEL
LIN {X 0,Y 278.601,Z 695.279,A -85,B 0,C 180,E1 -26398.534,E2 -26398.534} C_VEL
LIN {X 0,Y 285.838,Z 689.45,A -85,B 0,C 180,E1 -26400.971,E2 -26400.971} C_VEL
LIN {X 0,Y 293.838,Z 682.052,A -85,B 0,C 180,E1 -26403.248,E2 -26403.248} C_VEL
LIN {X 0,Y 301.312,Z 674.183,A -85,B 0,C 180,E1 -26405.124,E2 -26405.124} C_VEL
LIN {X 0,Y 309.341,Z 664.714,A -85,B 0,C 180,E1 -26406.873,E2 -26406.873} C_VEL
LIN {X 0,Y 316.556,Z 655.145,A -85,B 0,C 180,E1 -26408.284,E2 -26408.284} C_VEL
LIN {X 0,Y 324.194,Z 643.798,A -85,B 0,C 180,E1 -26409.596,E2 -26409.596} C_VEL
LIN {X 0,Y 331.46,Z 631.385,A -85,B 0,C 180,E1 -26410.727,E2 -26410.727} C_VEL
LIN {X 0,Y 338.459,Z 617.494,A -85,B 0,C 180,E1 -26411.703,E2 -26411.703} C_VEL
LIN {X 0,Y 344.786,Z 602.594,A -85,B 0,C 180,E1 -26412.492,E2 -26412.492} C_VEL
LIN {X 0,Y 350.584,Z 585.545,A -85,B 0,C 180,E1 -26413.18,E2 -26413.18} C_VEL
LIN {X 0,Y 364.529,Z 532.264,A -85,B 0,C 180,E1 -26414.951,E2 -26414.951} C_VEL
LIN {X 0,Y 364.541,Z 532.23,A -85,B 0,C 180,E1 -26415.017,E2 -26415.017} C_VEL
LIN {X 0,Y 350.49,Z 585.958,A -85,B 0,C 180,E1 -26416.806,E2 -26416.806} C_VEL
LIN {X 0,Y 344.519,Z 603.36,A -85,B 0,C 180,E1 -26417.513,E2 -26417.513} C_VEL
LIN {X 0,Y 338.906,Z 616.578,A -85,B 0,C 180,E1 -26418.245,E2 -26418.245} C_VEL
LIN {X 0,Y 332.175,Z 630.021,A -85,B 0,C 180,E1 -26419.18,E2 -26419.18} C_VEL
LIN {X 0,Y 324.339,Z 643.512,A -85,B 0,C 180,E1 -26420.426,E2 -26420.426} C_VEL
LIN {X 0,Y 316.754,Z 654.768,A -85,B 0,C 180,E1 -26421.745,E2 -26421.745} C_VEL
LIN {X 0,Y 308.4,Z 665.727,A -85,B 0,C 180,E1 -26423.402,E2 -26423.402} C_VEL
LIN {X 0,Y 300.495,Z 674.893,A -85,B 0,C 180,E1 -26425.174,E2 -26425.174} C_VEL
LIN {X 0,Y 294.102,Z 681.519,A -85,B 0,C 180,E1 -26426.786,E2 -26426.786} C_VEL
LIN {X 0,Y 286.175,Z 688.845,A -85,B 0,C 180,E1 -26429.07,E2 -26429.07} C_VEL
LIN {X 0,Y 278.898,Z 694.653,A -85,B 0,C 180,E1 -26431.499,E2 -26431.499} C_VEL
LIN {X 0,Y 272.409,Z 699.04,A -85,B 0,C 180,E1 -26434.08,E2 -26434.08} C_VEL
LIN {X 0,Y 266.656,Z 702.13,A -85,B 0,C 180,E1 -26436.796,E2 -26436.796} C_VEL
LIN {X 0,Y 261.818,Z 703.974,A -85,B 0,C 180,E1 -26439.648,E2 -26439.648} C_VEL
LIN {X 0,Y 257.852,Z 704.616,A -85,B 0,C 180,E1 -26442.614,E2 -26442.614} C_VEL
LIN {X 0,Y 254.605,Z 704.055,A -85,B 0,C 180,E1 -26445.665,E2 -26445.665} C_VEL
LIN {X 0,Y 252.466,Z 702.296,A -85,B 0,C 180,E1 -26448.802,E2 -26448.802} C_VEL
LIN {X 0,Y 251.227,Z 699.313,A -85,B 0,C 180,E1 -26451.987,E2 -26451.987} C_VEL
LIN {X 0,Y 250.726,Z 695.02,A -85,B 0,C 180,E1 -26455.193,E2 -26455.193} C_VEL
LIN {X 0,Y 250.912,Z 689.281,A -85,B 0,C 180,E1 -26458.401,E2 -26458.401} C_VEL
LIN {X 0,Y 251.163,Z 682.781,A -85,B 0,C 180,E1 -26461.199,E2 -26461.199} C_VEL
LIN {X 0,Y 251.45,Z 675.942,A -85,B 0,C 180,E1 -26463.594,E2 -26463.594} C_VEL
LIN {X 0,Y 251.601,Z 667.624,A -85,B 0,C 180,E1 -26465.993,E2 -26465.993} C_VEL
LIN {X 0,Y 252.052,Z 657.698,A -85,B 0,C 180,E1 -26468.39,E2 -26468.39} C_VEL
LIN {X 0,Y 252.471,Z 646.615,A -85,B 0,C 180,E1 -26470.592,E2 -26470.592} C_VEL
LIN {X 0,Y 253.229,Z 634.618,A -85,B 0,C 180,E1 -26472.582,E2 -26472.582} C_VEL
LIN {X 0,Y 253.957,Z 621.511,A -85,B 0,C 180,E1 -26474.373,E2 -26474.373} C_VEL
LIN {X 0,Y 254.842,Z 607.128,A -85,B 0,C 180,E1 -26475.954,E2 -26475.954} C_VEL
LIN {X 0,Y 255.562,Z 592.051,A -85,B 0,C 180,E1 -26477.239,E2 -26477.239} C_VEL
LIN {X 0,Y 256.258,Z 576.55,A -85,B 0,C 180,E1 -26478.218,E2 -26478.218} C_VEL
LIN {X 0,Y 259.843,Z 479.641,A -85,B 0,C 180,E1 -26482.993,E2 -26482.993} C_VEL
LIN {X 0,Y 257.791,Z 451.002,A -85,B 0,C 180,E1 -26484.399,E2 -26484.399} C_VEL
LIN {X 0,Y 257.593,Z 439.534,A -85,B 0,C 180,E1 -26484.982,E2 -26484.982} C_VEL
LIN {X 0,Y 260.557,Z 413.187,A -85,B 0,C 180,E1 -26489.824,E2 -26489.824} C_VEL
LIN {X 0,Y 261.539,Z 405.027,A -85,B 0,C 180,E1 -26491.313,E2 -26491.313} C_VEL
LIN {X 0,Y 258.554,Z 390.695,A -85,B 0,C 180,E1 -26494.148,E2 -26494.148} C_VEL
LIN {X 0,Y 254.183,Z 370.636,A -85,B 0,C 180,E1 -26498.246,E2 -26498.246} C_VEL
LIN {X 0,Y 253.222,Z 366.498,A -85,B 0,C 180,E1 -26499.161,E2 -26499.161} C_VEL
LIN {X 0,Y 253.18,Z 366.504,A -85,B 0,C 180,E1 -26504.002,E2 -26504.002} C_VEL
LIN {X 0,Y 253.175,Z 366.506,A -85,B 0,C 180,E1 -26508.395,E2 -26508.395} C_VEL
LIN {X 0,Y 253.146,Z 366.506,A -85,B 0,C 180,E1 -26512.502,E2 -26512.502} C_VEL
LIN {X 0,Y 253.222,Z 366.49,A -85,B 0,C 180,E1 -26516.412,E2 -26516.412} C_VEL
LIN {X 0,Y 253.18,Z 366.481,A -85,B 0,C 180,E1 -26518.945,E2 -26518.945} C_VEL
LIN {X 0,Y 254.181,Z 369.328,A -85,B 0,C 180,E1 -26519.214,E2 -26519.214} C_VEL
LIN {X 0,Y 255.814,Z 371.832,A -85,B 0,C 180,E1 -26519.547,E2 -26519.547} C_VEL
LIN {X 0,Y 264.86,Z 387.99,A -85,B 0,C 180,E1 -26521.365,E2 -26521.365} C_VEL
LIN {X 0,Y 272.278,Z 403.232,A -85,B 0,C 180,E1 -26522.801,E2 -26522.801} C_VEL
LIN {X 0,Y 275.847,Z 411.337,A -85,B 0,C 180,E1 -26523.481,E2 -26523.481} C_VEL
LIN {X 0,Y 273.961,Z 464.44,A -85,B 0,C 180,E1 -26524.821,E2 -26524.821} C_VEL
LIN {X 0,Y 273.423,Z 485.392,A -85,B 0,C 180,E1 -26525.445,E2 -26525.445} C_VEL
LIN {X 0,Y 272.654,Z 499.969,A -85,B 0,C 180,E1 -26526.183,E2 -26526.183} C_VEL
LIN {X 0,Y 271.342,Z 513.238,A -85,B 0,C 180,E1 -26527.119,E2 -26527.119} C_VEL
LIN {X 0,Y 269.688,Z 525.742,A -85,B 0,C 180,E1 -26528.278,E2 -26528.278} C_VEL
LIN {X 0,Y 267.908,Z 537.918,A -85,B 0,C 180,E1 -26529.732,E2 -26529.732} C_VEL
LIN {X 0,Y 265.658,Z 550.238,A -85,B 0,C 180,E1 -26531.555,E2 -26531.555} C_VEL
LIN {X 0,Y 263.275,Z 561.053,A -85,B 0,C 180,E1 -26533.535,E2 -26533.535} C_VEL
LIN {X 0,Y 260.977,Z 570.409,A -85,B 0,C 180,E1 -26535.625,E2 -26535.625} C_VEL
LIN {X 0,Y 258.918,Z 578.733,A -85,B 0,C 180,E1 -26537.898,E2 -26537.898} C_VEL
LIN {X 0,Y 256.9,Z 586.688,A -85,B 0,C 180,E1 -26540.585,E2 -26540.585} C_VEL
LIN {X 0,Y 255.372,Z 592.313,A -85,B 0,C 180,E1 -26542.91,E2 -26542.91} C_VEL
LIN {X 0,Y 253.988,Z 598.219,A -85,B 0,C 180,E1 -26546.047,E2 -26546.047} C_VEL
LIN {X 0,Y 253.196,Z 601.634,A -85,B 0,C 180,E1 -26548.415,E2 -26548.415} C_VEL
LIN {X 0,Y 252.601,Z 604.949,A -85,B 0,C 180,E1 -26551.589,E2 -26551.589} C_VEL
LIN {X 0,Y 252.615,Z 606.898,A -85,B 0,C 180,E1 -26554.772,E2 -26554.772} C_VEL
LIN {X 0,Y 252.9,Z 607.565,A -85,B 0,C 180,E1 -26557.96,E2 -26557.96} C_VEL
LIN {X 0,Y 253.681,Z 606.934,A -85,B 0,C 180,E1 -26561.144,E2 -26561.144} C_VEL
LIN {X 0,Y 255.015,Z 604.986,A -85,B 0,C 180,E1 -26564.312,E2 -26564.312} C_VEL
LIN {X 0,Y 257.034,Z 601.6,A -85,B 0,C 180,E1 -26567.485,E2 -26567.485} C_VEL
LIN {X 0,Y 259.483,Z 596.842,A -85,B 0,C 180,E1 -26570.544,E2 -26570.544} C_VEL
LIN {X 0,Y 262.504,Z 590.398,A -85,B 0,C 180,E1 -26573.594,E2 -26573.594} C_VEL
LIN {X 0,Y 265.346,Z 583.819,A -85,B 0,C 180,E1 -26576,E2 -26576} C_VEL
LIN {X 0,Y 268.609,Z 575.591,A -85,B 0,C 180,E1 -26578.418,E2 -26578.418} C_VEL
LIN {X 0,Y 271.965,Z 566.436,A -85,B 0,C 180,E1 -26580.575,E2 -26580.575} C_VEL
LIN {X 0,Y 275.311,Z 555.754,A -85,B 0,C 180,E1 -26582.617,E2 -26582.617} C_VEL
LIN {X 0,Y 278.275,Z 545.017,A -85,B 0,C 180,E1 -26584.278,E2 -26584.278} C_VEL
LIN {X 0,Y 281.328,Z 532.51,A -85,B 0,C 180,E1 -26585.81,E2 -26585.81} C_VEL
LIN {X 0,Y 283.504,Z 520.34,A -85,B 0,C 180,E1 -26587.03,E2 -26587.03} C_VEL
LIN {X 0,Y 285.369,Z 507.148,A -85,B 0,C 180,E1 -26588.049,E2 -26588.049} C_VEL
LIN {X 0,Y 286.753,Z 493.512,A -85,B 0,C 180,E1 -26588.82,E2 -26588.82} C_VEL
LIN {X 0,Y 287.524,Z 479.675,A -85,B 0,C 180,E1 -26589.352,E2 -26589.352} C_VEL
LIN {X 0,Y 289.679,Z 427.154,A -85,B 0,C 180,E1 -26590.654,E2 -26590.654} C_VEL
LIN {X 0,Y 281.471,Z 411.028,A -85,B 0,C 180,E1 -26592.531,E2 -26592.531} C_VEL
LIN {X 0,Y 273.275,Z 397.032,A -85,B 0,C 180,E1 -26594.505,E2 -26594.505} C_VEL
LIN {X 0,Y 267.382,Z 387.773,A -85,B 0,C 180,E1 -26596.012,E2 -26596.012} C_VEL
LIN {X 0,Y 261.249,Z 378.937,A -85,B 0,C 180,E1 -26597.668,E2 -26597.668} C_VEL
LIN {X 0,Y 258.999,Z 375.689,A -85,B 0,C 180,E1 -26598.308,E2 -26598.308} C_VEL
LIN {X 0,Y 256.739,Z 372.506,A -85,B 0,C 180,E1 -26598.967,E2 -26598.967} C_VEL
LIN {X 0,Y 255.953,Z 371.334,A -85,B 0,C 180,E1 -26599.203,E2 -26599.203} C_VEL
LIN {X 0,Y 253.954,Z 369.001,A -85,B 0,C 180,E1 -26599.79,E2 -26599.79} C_VEL
LIN {X 0,Y 253.141,Z 366.503,A -85,B 0,C 180,E1 -26600.153,E2 -26600.153} C_VEL
LIN {X 0,Y 253.165,Z 366.457,A -85,B 0,C 180,E1 -26604.477,E2 -26604.477} C_VEL
LIN {X 0,Y 253.157,Z 366.497,A -85,B 0,C 180,E1 -26608.284,E2 -26608.284} C_VEL
LIN {X 0,Y 253.184,Z 366.502,A -85,B 0,C 180,E1 -26612.289,E2 -26612.289} C_VEL
LIN {X 0,Y 253.342,Z 366.488,A -85,B 0,C 180,E1 -26615.839,E2 -26615.839} C_VEL
LIN {X 0,Y 257.745,Z 386.142,A -85,B 0,C 180,E1 -26616.846,E2 -26616.846} C_VEL
LIN {X 0,Y 258.944,Z 391.332,A -85,B 0,C 180,E1 -26617.106,E2 -26617.106} C_VEL
LIN {X 0,Y 256.586,Z 466.41,A -85,B 0,C 180,E1 -26620.67,E2 -26620.67} C_VEL
LIN {X 0,Y 256.094,Z 485.588,A -85,B 0,C 180,E1 -26621.667,E2 -26621.667} C_VEL
LIN {X 0,Y 255.492,Z 500.919,A -85,B 0,C 180,E1 -26622.756,E2 -26622.756} C_VEL
LIN {X 0,Y 254.668,Z 516.734,A -85,B 0,C 180,E1 -26624.249,E2 -26624.249} C_VEL
LIN {X 0,Y 253.936,Z 530.105,A -85,B 0,C 180,E1 -26625.829,E2 -26625.829} C_VEL
LIN {X 0,Y 253.241,Z 543.776,A -85,B 0,C 180,E1 -26627.824,E2 -26627.824} C_VEL
LIN {X 0,Y 252.499,Z 556.191,A -85,B 0,C 180,E1 -26630.015,E2 -26630.015} C_VEL
LIN {X 0,Y 251.97,Z 567.497,A -85,B 0,C 180,E1 -26632.412,E2 -26632.412} C_VEL
LIN {X 0,Y 251.738,Z 576.948,A -85,B 0,C 180,E1 -26634.811,E2 -26634.811} C_VEL
LIN {X 0,Y 251.759,Z 586.182,A -85,B 0,C 180,E1 -26637.608,E2 -26637.608} C_VEL
LIN {X 0,Y 252.103,Z 594.76,A -85,B 0,C 180,E1 -26640.796,E2 -26640.796} C_VEL
LIN {X 0,Y 253.114,Z 601.548,A -85,B 0,C 180,E1 -26643.967,E2 -26643.967} C_VEL
LIN {X 0,Y 254.547,Z 605.958,A -85,B 0,C 180,E1 -26646.533,E2 -26646.533} C_VEL
LIN {X 0,Y 254.696,Z 607.783,A -85,B 0,C 180,E1 -26647.8,E2 -26647.8} C_VEL
LIN {X 0,Y 253.415,Z 610.397,A -85,B 0,C 180,E1 -26649.939,E2 -26649.939} C_VEL
LIN {X 0,Y 252.557,Z 612.581,A -85,B 0,C 180,E1 -26652.12,E2 -26652.12} C_VEL
LIN {X 0,Y 253.358,Z 613.625,A -85,B 0,C 180,E1 -26653.422,E2 -26653.422} C_VEL
LIN {X 0,Y 256.642,Z 615.084,A -85,B 0,C 180,E1 -26655.838,E2 -26655.838} C_VEL
LIN {X 0,Y 261.673,Z 615.647,A -85,B 0,C 180,E1 -26658.736,E2 -26658.736} C_VEL
LIN {X 0,Y 267.184,Z 614.931,A -85,B 0,C 180,E1 -26661.532,E2 -26661.532} C_VEL
LIN {X 0,Y 273.296,Z 612.936,A -85,B 0,C 180,E1 -26664.209,E2 -26664.209} C_VEL
LIN {X 0,Y 280.059,Z 609.548,A -85,B 0,C 180,E1 -26666.756,E2 -26666.756} C_VEL
LIN {X 0,Y 287.41,Z 604.744,A -85,B 0,C 180,E1 -26669.171,E2 -26669.171} C_VEL
LIN {X 0,Y 295.234,Z 598.44,A -85,B 0,C 180,E1 -26671.463,E2 -26671.463} C_VEL
LIN {X 0,Y 302.557,Z 591.461,A -85,B 0,C 180,E1 -26673.355,E2 -26673.355} C_VEL
LIN {X 0,Y 310.538,Z 582.577,A -85,B 0,C 180,E1 -26675.21,E2 -26675.21} C_VEL
LIN {X 0,Y 318.244,Z 572.521,A -85,B 0,C 180,E1 -26676.853,E2 -26676.853} C_VEL
LIN {X 0,Y 325.911,Z 560.944,A -85,B 0,C 180,E1 -26678.358,E2 -26678.358} C_VEL
LIN {X 0,Y 333.095,Z 547.912,A -85,B 0,C 180,E1 -26679.697,E2 -26679.697} C_VEL
LIN {X 0,Y 338.589,Z 536.327,A -85,B 0,C 180,E1 -26680.666,E2 -26680.666} C_VEL
LIN {X 0,Y 343.468,Z 523.852,A -85,B 0,C 180,E1 -26681.512,E2 -26681.512} C_VEL
LIN {X 0,Y 348.193,Z 508.753,A -85,B 0,C 180,E1 -26682.323,E2 -26682.323} C_VEL
LIN {X 0,Y 352.902,Z 490.395,A -85,B 0,C 180,E1 -26683.115,E2 -26683.115} C_VEL
LIN {X 0,Y 352.843,Z 490.505,A -85,B 0,C 180,E1 -26683.492,E2 -26683.492} C_VEL
LIN {X 0,Y 349.206,Z 505.301,A -85,B 0,C 180,E1 -26684.641,E2 -26684.641} C_VEL
LIN {X 0,Y 347.706,Z 511.264,A -85,B 0,C 180,E1 -26684.959,E2 -26684.959} C_VEL
LIN {X 0,Y 342.347,Z 528.579,A -85,B 0,C 180,E1 -26685.584,E2 -26685.584} C_VEL
LIN {X 0,Y 336.598,Z 543.577,A -85,B 0,C 180,E1 -26686.218,E2 -26686.218} C_VEL
LIN {X 0,Y 329.022,Z 559.734,A -85,B 0,C 180,E1 -26687.059,E2 -26687.059} C_VEL
LIN {X 0,Y 320.948,Z 574.253,A -85,B 0,C 180,E1 -26688.067,E2 -26688.067} C_VEL
LIN {X 0,Y 313.227,Z 586.393,A -85,B 0,C 180,E1 -26689.148,E2 -26689.148} C_VEL
LIN {X 0,Y 303.86,Z 599.373,A -85,B 0,C 180,E1 -26690.66,E2 -26690.66} C_VEL
LIN {X 0,Y 295.088,Z 610.147,A -85,B 0,C 180,E1 -26692.322,E2 -26692.322} C_VEL
LIN {X 0,Y 285.72,Z 620.45,A -85,B 0,C 180,E1 -26694.392,E2 -26694.392} C_VEL
LIN {X 0,Y 278.304,Z 627.868,A -85,B 0,C 180,E1 -26696.378,E2 -26696.378} C_VEL
LIN {X 0,Y 270.569,Z 634.953,A -85,B 0,C 180,E1 -26698.818,E2 -26698.818} C_VEL
LIN {X 0,Y 263.74,Z 640.591,A -85,B 0,C 180,E1 -26701.442,E2 -26701.442} C_VEL
LIN {X 0,Y 257.908,Z 644.972,A -85,B 0,C 180,E1 -26704.244,E2 -26704.244} C_VEL
LIN {X 0,Y 253.043,Z 648.164,A -85,B 0,C 180,E1 -26707.199,E2 -26707.199} C_VEL
LIN {X 0,Y 249.323,Z 650.236,A -85,B 0,C 180,E1 -26710.298,E2 -26710.298} C_VEL
LIN {X 0,Y 246.838,Z 651.226,A -85,B 0,C 180,E1 -26713.515,E2 -26713.515} C_VEL
LIN {X 0,Y 246.056,Z 651.499,A -85,B 0,C 180,E1 -26714.944,E2 -26714.944} C_VEL
LIN {X 0,Y 244.789,Z 655.336,A -85,B 0,C 180,E1 -26717.607,E2 -26717.607} C_VEL
LIN {X 0,Y 244.498,Z 658.018,A -85,B 0,C 180,E1 -26720.102,E2 -26720.102} C_VEL
LIN {X 0,Y 244.911,Z 659.999,A -85,B 0,C 180,E1 -26722.502,E2 -26722.502} C_VEL
LIN {X 0,Y 244.689,Z 670.131,A -85,B 0,C 180,E1 -26725.073,E2 -26725.073} C_VEL
LIN {X 0,Y 244.534,Z 678.124,A -85,B 0,C 180,E1 -26727.537,E2 -26727.537} C_VEL
LIN {X 0,Y 244.362,Z 684.746,A -85,B 0,C 180,E1 -26730,E2 -26730} C_VEL
LIN {X 0,Y 244.036,Z 690.143,A -85,B 0,C 180,E1 -26732.467,E2 -26732.467} C_VEL
LIN {X 0,Y 243.912,Z 694.536,A -85,B 0,C 180,E1 -26734.942,E2 -26734.942} C_VEL
LIN {X 0,Y 244.245,Z 699.116,A -85,B 0,C 180,E1 -26738.244,E2 -26738.244} C_VEL
LIN {X 0,Y 245.439,Z 702.379,A -85,B 0,C 180,E1 -26741.523,E2 -26741.523} C_VEL
LIN {X 0,Y 247.54,Z 704.421,A -85,B 0,C 180,E1 -26744.754,E2 -26744.754} C_VEL
LIN {X 0,Y 250.833,Z 705.289,A -85,B 0,C 180,E1 -26747.889,E2 -26747.889} C_VEL
LIN {X 0,Y 254.91,Z 704.965,A -85,B 0,C 180,E1 -26750.929,E2 -26750.929} C_VEL
LIN {X 0,Y 259.761,Z 703.471,A -85,B 0,C 180,E1 -26753.858,E2 -26753.858} C_VEL
LIN {X 0,Y 265.747,Z 700.746,A -85,B 0,C 180,E1 -26756.62,E2 -26756.62} C_VEL
LIN {X 0,Y 272.5,Z 696.752,A -85,B 0,C 180,E1 -26759.234,E2 -26759.234} C_VEL
LIN {X 0,Y 279.951,Z 691.421,A -85,B 0,C 180,E1 -26761.697,E2 -26761.697} C_VEL
LIN {X 0,Y 288.165,Z 684.604,A -85,B 0,C 180,E1 -26763.991,E2 -26763.991} C_VEL
LIN {X 0,Y 295.838,Z 677.312,A -85,B 0,C 180,E1 -26765.873,E2 -26765.873} C_VEL
LIN {X 0,Y 304.035,Z 668.55,A -85,B 0,C 180,E1 -26767.627,E2 -26767.627} C_VEL
LIN {X 0,Y 312.711,Z 658.037,A -85,B 0,C 180,E1 -26769.255,E2 -26769.255} C_VEL
LIN {X 0,Y 321.191,Z 646.266,A -85,B 0,C 180,E1 -26770.655,E2 -26770.655} C_VEL
LIN {X 0,Y 328.774,Z 634.223,A -85,B 0,C 180,E1 -26771.784,E2 -26771.784} C_VEL
LIN {X 0,Y 335.634,Z 621.691,A -85,B 0,C 180,E1 -26772.68,E2 -26772.68} C_VEL
LIN {X 0,Y 341.575,Z 609.064,A -85,B 0,C 180,E1 -26773.39,E2 -26773.39} C_VEL
LIN {X 0,Y 347.913,Z 592.674,A -85,B 0,C 180,E1 -26774.094,E2 -26774.094} C_VEL
LIN {X 0,Y 353.159,Z 575.171,A -85,B 0,C 180,E1 -26774.707,E2 -26774.707} C_VEL
LIN {X 0,Y 355.248,Z 567.225,A -85,B 0,C 180,E1 -26774.967,E2 -26774.967} C_VEL
LIN {X 0,Y 355.272,Z 567.148,A -85,B 0,C 180,E1 -26775.009,E2 -26775.009} C_VEL
LIN {X 0,Y 349.272,Z 588.611,A -85,B 0,C 180,E1 -26775.722,E2 -26775.722} C_VEL
LIN {X 0,Y 343.677,Z 604.049,A -85,B 0,C 180,E1 -26776.338,E2 -26776.338} C_VEL
LIN {X 0,Y 337.426,Z 618.06,A -85,B 0,C 180,E1 -26777.098,E2 -26777.098} C_VEL
LIN {X 0,Y 330.484,Z 631.25,A -85,B 0,C 180,E1 -26777.999,E2 -26777.999} C_VEL
LIN {X 0,Y 322.664,Z 644.026,A -85,B 0,C 180,E1 -26779.16,E2 -26779.16} C_VEL
LIN {X 0,Y 314.18,Z 655.987,A -85,B 0,C 180,E1 -26780.551,E2 -26780.551} C_VEL
LIN {X 0,Y 305.511,Z 666.726,A -85,B 0,C 180,E1 -26782.172,E2 -26782.172} C_VEL
LIN {X 0,Y 297.299,Z 675.683,A -85,B 0,C 180,E1 -26783.914,E2 -26783.914} C_VEL
LIN {X 0,Y 290.598,Z 682.164,A -85,B 0,C 180,E1 -26785.498,E2 -26785.498} C_VEL
LIN {X 0,Y 282.268,Z 689.346,A -85,B 0,C 180,E1 -26787.757,E2 -26787.757} C_VEL
LIN {X 0,Y 274.625,Z 694.999,A -85,B 0,C 180,E1 -26790.174,E2 -26790.174} C_VEL
LIN {X 0,Y 269.367,Z 698.307,A -85,B 0,C 180,E1 -26792.092,E2 -26792.092} C_VEL
LIN {X 0,Y 263.081,Z 701.612,A -85,B 0,C 180,E1 -26794.787,E2 -26794.787} C_VEL
LIN {X 0,Y 257.251,Z 703.782,A -85,B 0,C 180,E1 -26797.782,E2 -26797.782} C_VEL
LIN {X 0,Y 253.069,Z 704.58,A -85,B 0,C 180,E1 -26800.602,E2 -26800.602} C_VEL
LIN {X 0,Y 249.305,Z 704.29,A -85,B 0,C 180,E1 -26803.683,E2 -26803.683} C_VEL
LIN {X 0,Y 246.553,Z 702.814,A -85,B 0,C 180,E1 -26806.864,E2 -26806.864} C_VEL
LIN {X 0,Y 244.676,Z 700.126,A -85,B 0,C 180,E1 -26810.11,E2 -26810.11} C_VEL
LIN {X 0,Y 243.989,Z 696.219,A -85,B 0,C 180,E1 -26813.406,E2 -26813.406} C_VEL
LIN {X 0,Y 243.813,Z 690.889,A -85,B 0,C 180,E1 -26816.707,E2 -26816.707} C_VEL
LIN {X 0,Y 244.084,Z 685.885,A -85,B 0,C 180,E1 -26819.178,E2 -26819.178} C_VEL
LIN {X 0,Y 244.299,Z 679.752,A -85,B 0,C 180,E1 -26821.643,E2 -26821.643} C_VEL
LIN {X 0,Y 244.531,Z 672.324,A -85,B 0,C 180,E1 -26824.107,E2 -26824.107} C_VEL
LIN {X 0,Y 244.744,Z 663.38,A -85,B 0,C 180,E1 -26826.574,E2 -26826.574} C_VEL
LIN {X 0,Y 245.244,Z 652.591,A -85,B 0,C 180,E1 -26829.038,E2 -26829.038} C_VEL
LIN {X 0,Y 245.921,Z 639.389,A -85,B 0,C 180,E1 -26831.501,E2 -26831.501} C_VEL
LIN {X 0,Y 246.613,Z 625.86,A -85,B 0,C 180,E1 -26833.552,E2 -26833.552} C_VEL
LIN {X 0,Y 247.544,Z 611.109,A -85,B 0,C 180,E1 -26835.336,E2 -26835.336} C_VEL
LIN {X 0,Y 248.292,Z 596.83,A -85,B 0,C 180,E1 -26836.703,E2 -26836.703} C_VEL
LIN {X 0,Y 248.911,Z 581.262,A -85,B 0,C 180,E1 -26837.82,E2 -26837.82} C_VEL
LIN {X 0,Y 250.422,Z 538.284,A -85,B 0,C 180,E1 -26840.092,E2 -26840.092} C_VEL
LIN {X 0,Y 252.753,Z 479.753,A -85,B 0,C 180,E1 -26843.054,E2 -26843.054} C_VEL
LIN {X 0,Y 250.729,Z 451.794,A -85,B 0,C 180,E1 -26844.474,E2 -26844.474} C_VEL
LIN {X 0,Y 250.526,Z 439.484,A -85,B 0,C 180,E1 -26845.128,E2 -26845.128} C_VEL
LIN {X 0,Y 253.553,Z 413.275,A -85,B 0,C 180,E1 -26850.047,E2 -26850.047} C_VEL
LIN {X 0,Y 254.479,Z 405.322,A -85,B 0,C 180,E1 -26851.532,E2 -26851.532} C_VEL
LIN {X 0,Y 250.307,Z 386.129,A -85,B 0,C 180,E1 -26855.438,E2 -26855.438} C_VEL
LIN {X 0,Y 246.181,Z 367.373,A -85,B 0,C 180,E1 -26859.441,E2 -26859.441} C_VEL
LIN {X 0,Y 246.118,Z 367.387,A -85,B 0,C 180,E1 -26863.082,E2 -26863.082} C_VEL
LIN {X 0,Y 246.118,Z 367.382,A -85,B 0,C 180,E1 -26866.919,E2 -26866.919} C_VEL
LIN {X 0,Y 246.109,Z 367.385,A -85,B 0,C 180,E1 -26871.234,E2 -26871.234} C_VEL
LIN {X 0,Y 246.147,Z 367.38,A -85,B 0,C 180,E1 -26875.613,E2 -26875.613} C_VEL
LIN {X 0,Y 246.139,Z 367.407,A -85,B 0,C 180,E1 -26877.86,E2 -26877.86} C_VEL
LIN {X 0,Y 247.018,Z 370.036,A -85,B 0,C 180,E1 -26878.098,E2 -26878.098} C_VEL
LIN {X 0,Y 248.735,Z 372.628,A -85,B 0,C 180,E1 -26878.468,E2 -26878.468} C_VEL
LIN {X 0,Y 257.471,Z 387.85,A -85,B 0,C 180,E1 -26880.32,E2 -26880.32} C_VEL
LIN {X 0,Y 264.815,Z 402.458,A -85,B 0,C 180,E1 -26881.812,E2 -26881.812} C_VEL
LIN {X 0,Y 269.545,Z 413.03,A -85,B 0,C 180,E1 -26882.754,E2 -26882.754} C_VEL
LIN {X 0,Y 267.674,Z 468.262,A -85,B 0,C 180,E1 -26884.196,E2 -26884.196} C_VEL
LIN {X 0,Y 267.131,Z 487.651,A -85,B 0,C 180,E1 -26884.816,E2 -26884.816} C_VEL
LIN {X 0,Y 266.247,Z 501.91,A -85,B 0,C 180,E1 -26885.573,E2 -26885.573} C_VEL
LIN {X 0,Y 264.766,Z 515.981,A -85,B 0,C 180,E1 -26886.62,E2 -26886.62} C_VEL
LIN {X 0,Y 262.942,Z 528.888,A -85,B 0,C 180,E1 -26887.897,E2 -26887.897} C_VEL
LIN {X 0,Y 260.906,Z 541.859,A -85,B 0,C 180,E1 -26889.574,E2 -26889.574} C_VEL
LIN {X 0,Y 258.537,Z 553.544,A -85,B 0,C 180,E1 -26891.438,E2 -26891.438} C_VEL
LIN {X 0,Y 255.942,Z 564.594,A -85,B 0,C 180,E1 -26893.618,E2 -26893.618} C_VEL
LIN {X 0,Y 253.464,Z 574.371,A -85,B 0,C 180,E1 -26896.007,E2 -26896.007} C_VEL
LIN {X 0,Y 251.141,Z 583.342,A -85,B 0,C 180,E1 -26898.742,E2 -26898.742} C_VEL
LIN {X 0,Y 249.36,Z 589.635,A -85,B 0,C 180,E1 -26901.113,E2 -26901.113} C_VEL
LIN {X 0,Y 248.041,Z 594.829,A -85,B 0,C 180,E1 -26903.514,E2 -26903.514} C_VEL
LIN {X 0,Y 246.696,Z 600.322,A -85,B 0,C 180,E1 -26906.745,E2 -26906.745} C_VEL
LIN {X 0,Y 245.738,Z 604.322,A -85,B 0,C 180,E1 -26910,E2 -26910} C_VEL
LIN {X 0,Y 245.517,Z 606.901,A -85,B 0,C 180,E1 -26913.271,E2 -26913.271} C_VEL
LIN {X 0,Y 245.669,Z 608.172,A -85,B 0,C 180,E1 -26916.549,E2 -26916.549} C_VEL
LIN {X 0,Y 246.263,Z 608.156,A -85,B 0,C 180,E1 -26919.826,E2 -26919.826} C_VEL
LIN {X 0,Y 247.308,Z 606.849,A -85,B 0,C 180,E1 -26923.096,E2 -26923.096} C_VEL
LIN {X 0,Y 249.177,Z 604.176,A -85,B 0,C 180,E1 -26926.326,E2 -26926.326} C_VEL
LIN {X 0,Y 251.472,Z 600.092,A -85,B 0,C 180,E1 -26929.527,E2 -26929.527} C_VEL
LIN {X 0,Y 254.355,Z 594.452,A -85,B 0,C 180,E1 -26932.677,E2 -26932.677} C_VEL
LIN {X 0,Y 257.376,Z 588.058,A -85,B 0,C 180,E1 -26935.381,E2 -26935.381} C_VEL
LIN {X 0,Y 260.757,Z 580.094,A -85,B 0,C 180,E1 -26938.04,E2 -26938.04} C_VEL
LIN {X 0,Y 264.052,Z 571.712,A -85,B 0,C 180,E1 -26940.266,E2 -26940.266} C_VEL
LIN {X 0,Y 267.685,Z 561.52,A -85,B 0,C 180,E1 -26942.441,E2 -26942.441} C_VEL
LIN {X 0,Y 270.863,Z 550.915,A -85,B 0,C 180,E1 -26944.29,E2 -26944.29} C_VEL
LIN {X 0,Y 273.798,Z 540.04,A -85,B 0,C 180,E1 -26945.818,E2 -26945.818} C_VEL
LIN {X 0,Y 276.615,Z 527.744,A -85,B 0,C 180,E1 -26947.198,E2 -26947.198} C_VEL
LIN {X 0,Y 278.696,Z 515.093,A -85,B 0,C 180,E1 -26948.351,E2 -26948.351} C_VEL
LIN {X 0,Y 280.434,Z 501.249,A -85,B 0,C 180,E1 -26949.297,E2 -26949.297} C_VEL
LIN {X 0,Y 281.597,Z 486.763,A -85,B 0,C 180,E1 -26949.992,E2 -26949.992} C_VEL
LIN {X 0,Y 282.466,Z 464.472,A -85,B 0,C 180,E1 -26950.633,E2 -26950.633} C_VEL
LIN {X 0,Y 284.031,Z 429.44,A -85,B 0,C 180,E1 -26951.497,E2 -26951.497} C_VEL
LIN {X 0,Y 276.327,Z 414.308,A -85,B 0,C 180,E1 -26953.338,E2 -26953.338} C_VEL
LIN {X 0,Y 267.378,Z 399.033,A -85,B 0,C 180,E1 -26955.602,E2 -26955.602} C_VEL
LIN {X 0,Y 260.649,Z 388.715,A -85,B 0,C 180,E1 -26957.425,E2 -26957.425} C_VEL
LIN {X 0,Y 255.238,Z 380.98,A -85,B 0,C 180,E1 -26958.986,E2 -26958.986} C_VEL
LIN {X 0,Y 252.166,Z 376.682,A -85,B 0,C 180,E1 -26959.919,E2 -26959.919} C_VEL
LIN {X 0,Y 249.929,Z 373.554,A -85,B 0,C 180,E1 -26960.625,E2 -26960.625} C_VEL
LIN {X 0,Y 249.044,Z 372.264,A -85,B 0,C 180,E1 -26960.912,E2 -26960.912} C_VEL
LIN {X 0,Y 246.986,Z 370.041,A -85,B 0,C 180,E1 -26961.562,E2 -26961.562} C_VEL
LIN {X 0,Y 246.067,Z 367.343,A -85,B 0,C 180,E1 -26961.998,E2 -26961.998} C_VEL
LIN {X 0,Y 246.119,Z 367.352,A -85,B 0,C 180,E1 -26965.623,E2 -26965.623} C_VEL
LIN {X 0,Y 246.123,Z 367.367,A -85,B 0,C 180,E1 -26969.185,E2 -26969.185} C_VEL
LIN {X 0,Y 246.141,Z 367.371,A -85,B 0,C 180,E1 -26972.914,E2 -26972.914} C_VEL
LIN {X 0,Y 246.309,Z 367.356,A -85,B 0,C 180,E1 -26975.751,E2 -26975.751} C_VEL
LIN {X 0,Y 250.234,Z 385.381,A -85,B 0,C 180,E1 -26976.721,E2 -26976.721} C_VEL
LIN {X 0,Y 251.846,Z 391.858,A -85,B 0,C 180,E1 -26977.054,E2 -26977.054} C_VEL
LIN {X 0,Y 249.552,Z 463.43,A -85,B 0,C 180,E1 -26980.583,E2 -26980.583} C_VEL
LIN {X 0,Y 249.039,Z 484.97,A -85,B 0,C 180,E1 -26981.712,E2 -26981.712} C_VEL
LIN {X 0,Y 248.404,Z 501.157,A -85,B 0,C 180,E1 -26982.883,E2 -26982.883} C_VEL
LIN {X 0,Y 247.595,Z 516.52,A -85,B 0,C 180,E1 -26984.368,E2 -26984.368} C_VEL
LIN {X 0,Y 246.85,Z 530.393,A -85,B 0,C 180,E1 -26986.043,E2 -26986.043} C_VEL
LIN {X 0,Y 246.128,Z 544.174,A -85,B 0,C 180,E1 -26988.092,E2 -26988.092} C_VEL
LIN {X 0,Y 245.413,Z 556.586,A -85,B 0,C 180,E1 -26990.346,E2 -26990.346} C_VEL
LIN {X 0,Y 244.935,Z 567.057,A -85,B 0,C 180,E1 -26992.606,E2 -26992.606} C_VEL
LIN {X 0,Y 244.7,Z 576.742,A -85,B 0,C 180,E1 -26995.073,E2 -26995.073} C_VEL
LIN {X 0,Y 244.747,Z 586.116,A -85,B 0,C 180,E1 -26997.949,E2 -26997.949} C_VEL
LIN {X 0,Y 245.029,Z 593.86,A -85,B 0,C 180,E1 -27000.819,E2 -27000.819} C_VEL
LIN {X 0,Y 245.959,Z 600.638,A -85,B 0,C 180,E1 -27003.88,E2 -27003.88} C_VEL
LIN {X 0,Y 247.881,Z 606.723,A -85,B 0,C 180,E1 -27007.305,E2 -27007.305} C_VEL
LIN {X 0,Y 249.635,Z 609.969,A -85,B 0,C 180,E1 -27009.692,E2 -27009.692} C_VEL
LIN {X 0,Y 252.631,Z 613.182,A -85,B 0,C 180,E1 -27012.815,E2 -27012.815} C_VEL
LIN {X 0,Y 253.358,Z 613.625,A -85,B 0,C 180,E1 -27013.422,E2 -27013.422} C_VEL
LIN {X 0,Y 254.371,Z 614.584,A -85,B 0,C 180,E1 -27014.72,E2 -27014.72} C_VEL
LIN {X 0,Y 254.855,Z 616.257,A -85,B 0,C 180,E1 -27017.816,E2 -27017.816} C_VEL
LIN {X 0,Y 255.967,Z 616.739,A -85,B 0,C 180,E1 -27019.564,E2 -27019.564} C_VEL
LIN {X 0,Y 257.244,Z 616.762,A -85,B 0,C 180,E1 -27020.392,E2 -27020.392} C_VEL
LIN {X 0,Y 260.73,Z 616.439,A -85,B 0,C 180,E1 -27022.092,E2 -27022.092} C_VEL
LIN {X 0,Y 267.052,Z 614.819,A -85,B 0,C 180,E1 -27024.813,E2 -27024.813} C_VEL
LIN {X 0,Y 274.033,Z 611.911,A -85,B 0,C 180,E1 -27027.393,E2 -27027.393} C_VEL
LIN {X 0,Y 281.61,Z 607.584,A -85,B 0,C 180,E1 -27029.832,E2 -27029.832} C_VEL
LIN {X 0,Y 289.704,Z 601.823,A -85,B 0,C 180,E1 -27032.135,E2 -27032.135} C_VEL
LIN {X 0,Y 298.344,Z 594.303,A -85,B 0,C 180,E1 -27034.296,E2 -27034.296} C_VEL
LIN {X 0,Y 306.292,Z 586.168,A -85,B 0,C 180,E1 -27036.076,E2 -27036.076} C_VEL
LIN {X 0,Y 314.583,Z 576.328,A -85,B 0,C 180,E1 -27037.756,E2 -27037.756} C_VEL
LIN {X 0,Y 321.831,Z 566.191,A -85,B 0,C 180,E1 -27039.136,E2 -27039.136} C_VEL
LIN {X 0,Y 329.95,Z 553.039,A -85,B 0,C 180,E1 -27040.551,E2 -27040.551} C_VEL
LIN {X 0,Y 336.181,Z 540.782,A -85,B 0,C 180,E1 -27041.615,E2 -27041.615} C_VEL
LIN {X 0,Y 341.91,Z 527.472,A -85,B 0,C 180,E1 -27042.535,E2 -27042.535} C_VEL
LIN {X 0,Y 346.767,Z 513.311,A -85,B 0,C 180,E1 -27043.326,E2 -27043.326} C_VEL
LIN {X 0,Y 348.249,Z 508.155,A -85,B 0,C 180,E1 -27043.556,E2 -27043.556} C_VEL
LIN {X 0,Y 346.992,Z 512.52,A -85,B 0,C 180,E1 -27043.815,E2 -27043.815} C_VEL
LIN {X 0,Y 341.847,Z 528.426,A -85,B 0,C 180,E1 -27044.369,E2 -27044.369} C_VEL
LIN {X 0,Y 335.582,Z 543.78,A -85,B 0,C 180,E1 -27045.004,E2 -27045.004} C_VEL
LIN {X 0,Y 327.805,Z 559.567,A -85,B 0,C 180,E1 -27045.803,E2 -27045.803} C_VEL
LIN {X 0,Y 319.527,Z 573.826,A -85,B 0,C 180,E1 -27046.761,E2 -27046.761} C_VEL
LIN {X 0,Y 310.846,Z 586.769,A -85,B 0,C 180,E1 -27047.904,E2 -27047.904} C_VEL
LIN {X 0,Y 302.568,Z 597.751,A -85,B 0,C 180,E1 -27049.157,E2 -27049.157} C_VEL
LIN {X 0,Y 293.346,Z 608.526,A -85,B 0,C 180,E1 -27050.745,E2 -27050.745} C_VEL
LIN {X 0,Y 284.741,Z 617.635,A -85,B 0,C 180,E1 -27052.494,E2 -27052.494} C_VEL
LIN {X 0,Y 276.764,Z 625.281,A -85,B 0,C 180,E1 -27054.402,E2 -27054.402} C_VEL
LIN {X 0,Y 268.408,Z 632.538,A -85,B 0,C 180,E1 -27056.768,E2 -27056.768} C_VEL
LIN {X 0,Y 260.949,Z 638.386,A -85,B 0,C 180,E1 -27059.336,E2 -27059.336} C_VEL
LIN {X 0,Y 254.457,Z 642.947,A -85,B 0,C 180,E1 -27062.098,E2 -27062.098} C_VEL
LIN {X 0,Y 248.83,Z 646.348,A -85,B 0,C 180,E1 -27065.023,E2 -27065.023} C_VEL
LIN {X 0,Y 244.394,Z 648.635,A -85,B 0,C 180,E1 -27068.124,E2 -27068.124} C_VEL
LIN {X 0,Y 241.236,Z 649.868,A -85,B 0,C 180,E1 -27071.373,E2 -27071.373} C_VEL
LIN {X 0,Y 239.448,Z 650.18,A -85,B 0,C 180,E1 -27074.083,E2 -27074.083} C_VEL
LIN {X 0,Y 237.821,Z 654.633,A -85,B 0,C 180,E1 -27077.238,E2 -27077.238} C_VEL
LIN {X 0,Y 237.434,Z 657.297,A -85,B 0,C 180,E1 -27079.804,E2 -27079.804} C_VEL
LIN {X 0,Y 237.955,Z 659.58,A -85,B 0,C 180,E1 -27082.919,E2 -27082.919} C_VEL
LIN {X 0,Y 237.789,Z 668.99,A -85,B 0,C 180,E1 -27085.353,E2 -27085.353} C_VEL
LIN {X 0,Y 237.631,Z 677.125,A -85,B 0,C 180,E1 -27087.888,E2 -27087.888} C_VEL
LIN {X 0,Y 237.409,Z 684.805,A -85,B 0,C 180,E1 -27090.845,E2 -27090.845} C_VEL
LIN {X 0,Y 237.077,Z 690.13,A -85,B 0,C 180,E1 -27093.387,E2 -27093.387} C_VEL
LIN {X 0,Y 237.063,Z 695.755,A -85,B 0,C 180,E1 -27096.787,E2 -27096.787} C_VEL
LIN {X 0,Y 237.675,Z 699.948,A -85,B 0,C 180,E1 -27100.185,E2 -27100.185} C_VEL
LIN {X 0,Y 239.522,Z 702.929,A -85,B 0,C 180,E1 -27103.529,E2 -27103.529} C_VEL
LIN {X 0,Y 242.337,Z 704.713,A -85,B 0,C 180,E1 -27106.8,E2 -27106.8} C_VEL
LIN {X 0,Y 246.12,Z 705.321,A -85,B 0,C 180,E1 -27109.969,E2 -27109.969} C_VEL
LIN {X 0,Y 250.643,Z 704.762,A -85,B 0,C 180,E1 -27113.032,E2 -27113.032} C_VEL
LIN {X 0,Y 256.291,Z 703.038,A -85,B 0,C 180,E1 -27115.93,E2 -27115.93} C_VEL
LIN {X 0,Y 262.904,Z 700.097,A -85,B 0,C 180,E1 -27118.657,E2 -27118.657} C_VEL
LIN {X 0,Y 270.174,Z 695.915,A -85,B 0,C 180,E1 -27121.232,E2 -27121.232} C_VEL
LIN {X 0,Y 278.201,Z 690.389,A -85,B 0,C 180,E1 -27123.635,E2 -27123.635} C_VEL
LIN {X 0,Y 286.972,Z 683.368,A -85,B 0,C 180,E1 -27125.859,E2 -27125.859} C_VEL
LIN {X 0,Y 295.164,Z 675.83,A -85,B 0,C 180,E1 -27127.666,E2 -27127.666} C_VEL
LIN {X 0,Y 303.791,Z 666.818,A -85,B 0,C 180,E1 -27129.35,E2 -27129.35} C_VEL
LIN {X 0,Y 312.896,Z 655.998,A -85,B 0,C 180,E1 -27130.903,E2 -27130.903} C_VEL
LIN {X 0,Y 321.221,Z 644.733,A -85,B 0,C 180,E1 -27132.15,E2 -27132.15} C_VEL
LIN {X 0,Y 328.954,Z 632.754,A -85,B 0,C 180,E1 -27133.192,E2 -27133.192} C_VEL
LIN {X 0,Y 336.928,Z 618.209,A -85,B 0,C 180,E1 -27134.142,E2 -27134.142} C_VEL
LIN {X 0,Y 343.522,Z 603.89,A -85,B 0,C 180,E1 -27134.842,E2 -27134.842} C_VEL
LIN {X 0,Y 343.413,Z 604.145,A -85,B 0,C 180,E1 -27135.128,E2 -27135.128} C_VEL
LIN {X 0,Y 337.654,Z 616.78,A -85,B 0,C 180,E1 -27135.771,E2 -27135.771} C_VEL
LIN {X 0,Y 329.783,Z 631.309,A -85,B 0,C 180,E1 -27136.712,E2 -27136.712} C_VEL
LIN {X 0,Y 322.6,Z 642.681,A -85,B 0,C 180,E1 -27137.694,E2 -27137.694} C_VEL
LIN {X 0,Y 314.432,Z 653.993,A -85,B 0,C 180,E1 -27138.917,E2 -27138.917} C_VEL
LIN {X 0,Y 306.604,Z 663.567,A -85,B 0,C 180,E1 -27140.233,E2 -27140.233} C_VEL
LIN {X 0,Y 297.83,Z 673.01,A -85,B 0,C 180,E1 -27141.877,E2 -27141.877} C_VEL
LIN {X 0,Y 288.405,Z 681.898,A -85,B 0,C 180,E1 -27143.917,E2 -27143.917} C_VEL
LIN {X 0,Y 280.673,Z 688.265,A -85,B 0,C 180,E1 -27145.84,E2 -27145.84} C_VEL
LIN {X 0,Y 272.608,Z 694.032,A -85,B 0,C 180,E1 -27148.149,E2 -27148.149} C_VEL
LIN {X 0,Y 265.938,Z 698.075,A -85,B 0,C 180,E1 -27150.363,E2 -27150.363} C_VEL
LIN {X 0,Y 259.881,Z 701.137,A -85,B 0,C 180,E1 -27152.73,E2 -27152.73} C_VEL
LIN {X 0,Y 253.752,Z 703.435,A -85,B 0,C 180,E1 -27155.541,E2 -27155.541} C_VEL
LIN {X 0,Y 248.581,Z 704.551,A -85,B 0,C 180,E1 -27158.512,E2 -27158.512} C_VEL
LIN {X 0,Y 244.356,Z 704.503,A -85,B 0,C 180,E1 -27161.621,E2 -27161.621} C_VEL
LIN {X 0,Y 240.883,Z 703.272,A -85,B 0,C 180,E1 -27164.829,E2 -27164.829} C_VEL
LIN {X 0,Y 238.613,Z 700.877,A -85,B 0,C 180,E1 -27168.143,E2 -27168.143} C_VEL
LIN {X 0,Y 237.307,Z 697.275,A -85,B 0,C 180,E1 -27171.514,E2 -27171.514} C_VEL
LIN {X 0,Y 236.86,Z 692.367,A -85,B 0,C 180,E1 -27174.911,E2 -27174.911} C_VEL
LIN {X 0,Y 237.102,Z 685.963,A -85,B 0,C 180,E1 -27178.308,E2 -27178.308} C_VEL
LIN {X 0,Y 237.35,Z 679.91,A -85,B 0,C 180,E1 -27180.846,E2 -27180.846} C_VEL
LIN {X 0,Y 237.612,Z 672.628,A -85,B 0,C 180,E1 -27183.38,E2 -27183.38} C_VEL
LIN {X 0,Y 237.803,Z 663.778,A -85,B 0,C 180,E1 -27185.918,E2 -27185.918} C_VEL
LIN {X 0,Y 238.283,Z 652.184,A -85,B 0,C 180,E1 -27188.665,E2 -27188.665} C_VEL
LIN {X 0,Y 238.841,Z 640.164,A -85,B 0,C 180,E1 -27190.99,E2 -27190.99} C_VEL
LIN {X 0,Y 239.539,Z 626.885,A -85,B 0,C 180,E1 -27193.099,E2 -27193.099} C_VEL
LIN {X 0,Y 240.306,Z 613.896,A -85,B 0,C 180,E1 -27194.777,E2 -27194.777} C_VEL
LIN {X 0,Y 241.049,Z 600.492,A -85,B 0,C 180,E1 -27196.176,E2 -27196.176} C_VEL
LIN {X 0,Y 241.729,Z 584.833,A -85,B 0,C 180,E1 -27197.442,E2 -27197.442} C_VEL
LIN {X 0,Y 242.522,Z 563.102,A -85,B 0,C 180,E1 -27198.688,E2 -27198.688} C_VEL
LIN {X 0,Y 245.611,Z 479.612,A -85,B 0,C 180,E1 -27203.122,E2 -27203.122} C_VEL
LIN {X 0,Y 243.574,Z 449.99,A -85,B 0,C 180,E1 -27204.672,E2 -27204.672} C_VEL
LIN {X 0,Y 243.455,Z 439.624,A -85,B 0,C 180,E1 -27205.225,E2 -27205.225} C_VEL
LIN {X 0,Y 246.41,Z 414.442,A -85,B 0,C 180,E1 -27210.067,E2 -27210.067} C_VEL
LIN {X 0,Y 247.29,Z 407.182,A -85,B 0,C 180,E1 -27211.454,E2 -27211.454} C_VEL
LIN {X 0,Y 246.942,Z 403.962,A -85,B 0,C 180,E1 -27212.099,E2 -27212.099} C_VEL
LIN {X 0,Y 242.063,Z 381.558,A -85,B 0,C 180,E1 -27216.782,E2 -27216.782} C_VEL
LIN {X 0,Y 239.137,Z 368.249,A -85,B 0,C 180,E1 -27219.696,E2 -27219.696} C_VEL
LIN {X 0,Y 239.084,Z 368.255,A -85,B 0,C 180,E1 -27224.679,E2 -27224.679} C_VEL
LIN {X 0,Y 239.072,Z 368.263,A -85,B 0,C 180,E1 -27227.634,E2 -27227.634} C_VEL
LIN {X 0,Y 239.063,Z 368.262,A -85,B 0,C 180,E1 -27232.288,E2 -27232.288} C_VEL
LIN {X 0,Y 239.098,Z 368.367,A -85,B 0,C 180,E1 -27236.676,E2 -27236.676} C_VEL
LIN {X 0,Y 240.019,Z 371.013,A -85,B 0,C 180,E1 -27236.937,E2 -27236.937} C_VEL
LIN {X 0,Y 241.792,Z 373.646,A -85,B 0,C 180,E1 -27237.343,E2 -27237.343} C_VEL
LIN {X 0,Y 249.717,Z 387.114,A -85,B 0,C 180,E1 -27239.123,E2 -27239.123} C_VEL
LIN {X 0,Y 257.38,Z 401.718,A -85,B 0,C 180,E1 -27240.759,E2 -27240.759} C_VEL
LIN {X 0,Y 263.387,Z 414.979,A -85,B 0,C 180,E1 -27242.013,E2 -27242.013} C_VEL
LIN {X 0,Y 261.501,Z 469.245,A -85,B 0,C 180,E1 -27243.463,E2 -27243.463} C_VEL
LIN {X 0,Y 260.932,Z 488.055,A -85,B 0,C 180,E1 -27244.073,E2 -27244.073} C_VEL
LIN {X 0,Y 260.027,Z 502.346,A -85,B 0,C 180,E1 -27244.843,E2 -27244.843} C_VEL
LIN {X 0,Y 258.482,Z 516.503,A -85,B 0,C 180,E1 -27245.91,E2 -27245.91} C_VEL
LIN {X 0,Y 256.722,Z 528.624,A -85,B 0,C 180,E1 -27247.12,E2 -27247.12} C_VEL
LIN {X 0,Y 254.813,Z 540.537,A -85,B 0,C 180,E1 -27248.64,E2 -27248.64} C_VEL
LIN {X 0,Y 252.403,Z 552.609,A -85,B 0,C 180,E1 -27250.548,E2 -27250.548} C_VEL
LIN {X 0,Y 249.973,Z 562.635,A -85,B 0,C 180,E1 -27252.48,E2 -27252.48} C_VEL
LIN {X 0,Y 247.392,Z 572.506,A -85,B 0,C 180,E1 -27254.818,E2 -27254.818} C_VEL
LIN {X 0,Y 245.2,Z 580.735,A -85,B 0,C 180,E1 -27257.21,E2 -27257.21} C_VEL
LIN {X 0,Y 243.044,Z 588.601,A -85,B 0,C 180,E1 -27260.043,E2 -27260.043} C_VEL
LIN {X 0,Y 241.422,Z 594.171,A -85,B 0,C 180,E1 -27262.498,E2 -27262.498} C_VEL
LIN {X 0,Y 239.962,Z 599.984,A -85,B 0,C 180,E1 -27265.815,E2 -27265.815} C_VEL
LIN {X 0,Y 239.074,Z 603.374,A -85,B 0,C 180,E1 -27268.321,E2 -27268.321} C_VEL
LIN {X 0,Y 238.512,Z 606.609,A -85,B 0,C 180,E1 -27271.683,E2 -27271.683} C_VEL
LIN {X 0,Y 238.539,Z 608.485,A -85,B 0,C 180,E1 -27275.054,E2 -27275.054} C_VEL
LIN {X 0,Y 238.892,Z 609.087,A -85,B 0,C 180,E1 -27278.43,E2 -27278.43} C_VEL
LIN {X 0,Y 239.786,Z 608.396,A -85,B 0,C 180,E1 -27281.799,E2 -27281.799} C_VEL
LIN {X 0,Y 241.326,Z 606.383,A -85,B 0,C 180,E1 -27285.143,E2 -27285.143} C_VEL
LIN {X 0,Y 243.483,Z 602.99,A -85,B 0,C 180,E1 -27288.448,E2 -27288.448} C_VEL
LIN {X 0,Y 246.225,Z 598.11,A -85,B 0,C 180,E1 -27291.705,E2 -27291.705} C_VEL
LIN {X 0,Y 249.524,Z 591.59,A -85,B 0,C 180,E1 -27294.902,E2 -27294.902} C_VEL
LIN {X 0,Y 252.802,Z 584.55,A -85,B 0,C 180,E1 -27297.546,E2 -27297.546} C_VEL
LIN {X 0,Y 256.194,Z 576.595,A -85,B 0,C 180,E1 -27299.932,E2 -27299.932} C_VEL
LIN {X 0,Y 259.835,Z 567.303,A -85,B 0,C 180,E1 -27302.169,E2 -27302.169} C_VEL
LIN {X 0,Y 263.508,Z 556.07,A -85,B 0,C 180,E1 -27304.362,E2 -27304.362} C_VEL
LIN {X 0,Y 266.99,Z 544.271,A -85,B 0,C 180,E1 -27306.178,E2 -27306.178} C_VEL
LIN {X 0,Y 269.926,Z 532.819,A -85,B 0,C 180,E1 -27307.577,E2 -27307.577} C_VEL
LIN {X 0,Y 272.26,Z 520.329,A -85,B 0,C 180,E1 -27308.837,E2 -27308.837} C_VEL
LIN {X 0,Y 274.26,Z 506.597,A -85,B 0,C 180,E1 -27309.894,E2 -27309.894} C_VEL
LIN {X 0,Y 275.72,Z 492.36,A -85,B 0,C 180,E1 -27310.676,E2 -27310.676} C_VEL
LIN {X 0,Y 276.419,Z 477.512,A -85,B 0,C 180,E1 -27311.212,E2 -27311.212} C_VEL
LIN {X 0,Y 278.517,Z 431.914,A -85,B 0,C 180,E1 -27312.356,E2 -27312.356} C_VEL
LIN {X 0,Y 271.331,Z 417.824,A -85,B 0,C 180,E1 -27314.15,E2 -27314.15} C_VEL
LIN {X 0,Y 262.785,Z 403.122,A -85,B 0,C 180,E1 -27316.411,E2 -27316.411} C_VEL
LIN {X 0,Y 254.753,Z 390.726,A -85,B 0,C 180,E1 -27318.708,E2 -27318.708} C_VEL
LIN {X 0,Y 248.456,Z 381.964,A -85,B 0,C 180,E1 -27320.65,E2 -27320.65} C_VEL
LIN {X 0,Y 245.593,Z 377.934,A -85,B 0,C 180,E1 -27321.595,E2 -27321.595} C_VEL
LIN {X 0,Y 243.24,Z 374.952,A -85,B 0,C 180,E1 -27322.387,E2 -27322.387} C_VEL
LIN {X 0,Y 242.316,Z 373.335,A -85,B 0,C 180,E1 -27322.727,E2 -27322.727} C_VEL
LIN {X 0,Y 240.135,Z 371.171,A -85,B 0,C 180,E1 -27323.471,E2 -27323.471} C_VEL
LIN {X 0,Y 239.143,Z 368.867,A -85,B 0,C 180,E1 -27323.881,E2 -27323.881} C_VEL
LIN {X 0,Y 239.022,Z 368.213,A -85,B 0,C 180,E1 -27323.989,E2 -27323.989} C_VEL
LIN {X 0,Y 239.079,Z 368.251,A -85,B 0,C 180,E1 -27328.172,E2 -27328.172} C_VEL
LIN {X 0,Y 239.099,Z 368.257,A -85,B 0,C 180,E1 -27332.048,E2 -27332.048} C_VEL
LIN {X 0,Y 239.254,Z 368.233,A -85,B 0,C 180,E1 -27335.694,E2 -27335.694} C_VEL
LIN {X 0,Y 242.814,Z 384.803,A -85,B 0,C 180,E1 -27336.612,E2 -27336.612} C_VEL
LIN {X 0,Y 244.69,Z 393.078,A -85,B 0,C 180,E1 -27337.052,E2 -27337.052} C_VEL
LIN {X 0,Y 242.46,Z 463.308,A -85,B 0,C 180,E1 -27340.651,E2 -27340.651} C_VEL
LIN {X 0,Y 241.891,Z 486.378,A -85,B 0,C 180,E1 -27341.917,E2 -27341.917} C_VEL
LIN {X 0,Y 241.236,Z 502.353,A -85,B 0,C 180,E1 -27343.12,E2 -27343.12} C_VEL
LIN {X 0,Y 240.566,Z 515.656,A -85,B 0,C 180,E1 -27344.429,E2 -27344.429} C_VEL
LIN {X 0,Y 239.78,Z 530.581,A -85,B 0,C 180,E1 -27346.269,E2 -27346.269} C_VEL
LIN {X 0,Y 239.103,Z 543.169,A -85,B 0,C 180,E1 -27348.166,E2 -27348.166} C_VEL
LIN {X 0,Y 238.394,Z 555.872,A -85,B 0,C 180,E1 -27350.486,E2 -27350.486} C_VEL
LIN {X 0,Y 237.914,Z 566.516,A -85,B 0,C 180,E1 -27352.812,E2 -27352.812} C_VEL
LIN {X 0,Y 237.674,Z 576.366,A -85,B 0,C 180,E1 -27355.351,E2 -27355.351} C_VEL
LIN {X 0,Y 237.723,Z 584.708,A -85,B 0,C 180,E1 -27357.889,E2 -27357.889} C_VEL
LIN {X 0,Y 237.984,Z 592.83,A -85,B 0,C 180,E1 -27360.843,E2 -27360.843} C_VEL
LIN {X 0,Y 238.992,Z 600.455,A -85,B 0,C 180,E1 -27364.201,E2 -27364.201} C_VEL
LIN {X 0,Y 240.86,Z 606.445,A -85,B 0,C 180,E1 -27367.519,E2 -27367.519} C_VEL
LIN {X 0,Y 242.652,Z 610.028,A -85,B 0,C 180,E1 -27369.973,E2 -27369.973} C_VEL
LIN {X 0,Y 245.736,Z 613.599,A -85,B 0,C 180,E1 -27373.181,E2 -27373.181} C_VEL
LIN {X 0,Y 249.863,Z 615.848,A -85,B 0,C 180,E1 -27376.28,E2 -27376.28} C_VEL
LIN {X 0,Y 255.032,Z 616.771,A -85,B 0,C 180,E1 -27379.243,E2 -27379.243} C_VEL
LIN {X 0,Y 257.244,Z 616.762,A -85,B 0,C 180,E1 -27380.392,E2 -27380.392} C_VEL
LIN {X 0,Y 259.081,Z 616.798,A -85,B 0,C 180,E1 -27381.64,E2 -27381.64} C_VEL
LIN {X 0,Y 260.733,Z 616.801,A -85,B 0,C 180,E1 -27383.798,E2 -27383.798} C_VEL
LIN {X 0,Y 262.767,Z 616.198,A -85,B 0,C 180,E1 -27385.909,E2 -27385.909} C_VEL
LIN {X 0,Y 265.144,Z 615.29,A -85,B 0,C 180,E1 -27387.059,E2 -27387.059} C_VEL
LIN {X 0,Y 271.89,Z 612.44,A -85,B 0,C 180,E1 -27389.306,E2 -27389.306} C_VEL
LIN {X 0,Y 279.318,Z 608.302,A -85,B 0,C 180,E1 -27391.502,E2 -27391.502} C_VEL
LIN {X 0,Y 288.529,Z 601.839,A -85,B 0,C 180,E1 -27393.942,E2 -27393.942} C_VEL
LIN {X 0,Y 297.66,Z 594.063,A -85,B 0,C 180,E1 -27396.036,E2 -27396.036} C_VEL
LIN {X 0,Y 306.07,Z 585.66,A -85,B 0,C 180,E1 -27397.747,E2 -27397.747} C_VEL
LIN {X 0,Y 314.69,Z 575.461,A -85,B 0,C 180,E1 -27399.372,E2 -27399.372} C_VEL
LIN {X 0,Y 322.335,Z 565.026,A -85,B 0,C 180,E1 -27400.686,E2 -27400.686} C_VEL
LIN {X 0,Y 330.682,Z 551.412,A -85,B 0,C 180,E1 -27402.057,E2 -27402.057} C_VEL
LIN {X 0,Y 336.559,Z 540.077,A -85,B 0,C 180,E1 -27402.968,E2 -27402.968} C_VEL
LIN {X 0,Y 338.448,Z 535.945,A -85,B 0,C 180,E1 -27403.258,E2 -27403.258} C_VEL
LIN {X 0,Y 337.901,Z 537.266,A -85,B 0,C 180,E1 -27403.487,E2 -27403.487} C_VEL
LIN {X 0,Y 330.009,Z 553.786,A -85,B 0,C 180,E1 -27404.246,E2 -27404.246} C_VEL
LIN {X 0,Y 322.151,Z 567.543,A -85,B 0,C 180,E1 -27405.037,E2 -27405.037} C_VEL
LIN {X 0,Y 313.046,Z 581.297,A -85,B 0,C 180,E1 -27406.081,E2 -27406.081} C_VEL
LIN {X 0,Y 304.318,Z 592.816,A -85,B 0,C 180,E1 -27407.234,E2 -27407.234} C_VEL
LIN {X 0,Y 294.593,Z 604.178,A -85,B 0,C 180,E1 -27408.715,E2 -27408.715} C_VEL
LIN {X 0,Y 285.446,Z 613.698,A -85,B 0,C 180,E1 -27410.356,E2 -27410.356} C_VEL
LIN {X 0,Y 275.623,Z 622.811,A -85,B 0,C 180,E1 -27412.416,E2 -27412.416} C_VEL
LIN {X 0,Y 266.705,Z 630.206,A -85,B 0,C 180,E1 -27414.705,E2 -27414.705} C_VEL
LIN {X 0,Y 258.576,Z 636.237,A -85,B 0,C 180,E1 -27417.195,E2 -27417.195} C_VEL
LIN {X 0,Y 251.377,Z 640.98,A -85,B 0,C 180,E1 -27419.897,E2 -27419.897} C_VEL
LIN {X 0,Y 245.235,Z 644.563,A -85,B 0,C 180,E1 -27422.806,E2 -27422.806} C_VEL
LIN {X 0,Y 240.033,Z 647.043,A -85,B 0,C 180,E1 -27425.887,E2 -27425.887} C_VEL
LIN {X 0,Y 236.022,Z 648.433,A -85,B 0,C 180,E1 -27429.137,E2 -27429.137} C_VEL
LIN {X 0,Y 232.944,Z 648.817,A -85,B 0,C 180,E1 -27433.177,E2 -27433.177} C_VEL
LIN {X 0,Y 231.171,Z 652.85,A -85,B 0,C 180,E1 -27435.971,E2 -27435.971} C_VEL
LIN {X 0,Y 230.356,Z 656.573,A -85,B 0,C 180,E1 -27439.488,E2 -27439.488} C_VEL
LIN {X 0,Y 231.064,Z 659.347,A -85,B 0,C 180,E1 -27443.418,E2 -27443.418} C_VEL
LIN {X 0,Y 230.915,Z 669.243,A -85,B 0,C 180,E1 -27446.086,E2 -27446.086} C_VEL
LIN {X 0,Y 230.714,Z 677.243,A -85,B 0,C 180,E1 -27448.695,E2 -27448.695} C_VEL
LIN {X 0,Y 230.552,Z 682.816,A -85,B 0,C 180,E1 -27450.87,E2 -27450.87} C_VEL
LIN {X 0,Y 230.224,Z 688.384,A -85,B 0,C 180,E1 -27453.488,E2 -27453.488} C_VEL
LIN {X 0,Y 230.175,Z 694.329,A -85,B 0,C 180,E1 -27456.991,E2 -27456.991} C_VEL
LIN {X 0,Y 230.786,Z 698.836,A -85,B 0,C 180,E1 -27460.492,E2 -27460.492} C_VEL
LIN {X 0,Y 232.654,Z 702.134,A -85,B 0,C 180,E1 -27463.937,E2 -27463.937} C_VEL
LIN {X 0,Y 235.575,Z 704.249,A -85,B 0,C 180,E1 -27467.297,E2 -27467.297} C_VEL
LIN {X 0,Y 239.94,Z 705.24,A -85,B 0,C 180,E1 -27470.908,E2 -27470.908} C_VEL
LIN {X 0,Y 244.142,Z 705.032,A -85,B 0,C 180,E1 -27473.682,E2 -27473.682} C_VEL
LIN {X 0,Y 249.967,Z 703.71,A -85,B 0,C 180,E1 -27476.637,E2 -27476.637} C_VEL
LIN {X 0,Y 256.768,Z 701.197,A -85,B 0,C 180,E1 -27479.408,E2 -27479.408} C_VEL
LIN {X 0,Y 265.157,Z 696.944,A -85,B 0,C 180,E1 -27482.294,E2 -27482.294} C_VEL
LIN {X 0,Y 272.5,Z 692.438,A -85,B 0,C 180,E1 -27484.437,E2 -27484.437} C_VEL
LIN {X 0,Y 281.48,Z 685.963,A -85,B 0,C 180,E1 -27486.671,E2 -27486.671} C_VEL
LIN {X 0,Y 289.878,Z 679.007,A -85,B 0,C 180,E1 -27488.477,E2 -27488.477} C_VEL
LIN {X 0,Y 298.682,Z 670.689,A -85,B 0,C 180,E1 -27490.159,E2 -27490.159} C_VEL
LIN {X 0,Y 307.963,Z 660.711,A -85,B 0,C 180,E1 -27491.703,E2 -27491.703} C_VEL
LIN {X 0,Y 316.416,Z 650.369,A -85,B 0,C 180,E1 -27492.943,E2 -27492.943} C_VEL
LIN {X 0,Y 325.612,Z 637.434,A -85,B 0,C 180,E1 -27494.142,E2 -27494.142} C_VEL
LIN {X 0,Y 331.918,Z 627.241,A -85,B 0,C 180,E1 -27494.86,E2 -27494.86} C_VEL
LIN {X 0,Y 331.729,Z 627.556,A -85,B 0,C 180,E1 -27495.159,E2 -27495.159} C_VEL
LIN {X 0,Y 324.231,Z 639.474,A -85,B 0,C 180,E1 -27496.052,E2 -27496.052} C_VEL
LIN {X 0,Y 314.692,Z 652.555,A -85,B 0,C 180,E1 -27497.351,E2 -27497.351} C_VEL
LIN {X 0,Y 305.505,Z 663.444,A -85,B 0,C 180,E1 -27498.764,E2 -27498.764} C_VEL
LIN {X 0,Y 296.379,Z 672.856,A -85,B 0,C 180,E1 -27500.35,E2 -27500.35} C_VEL
LIN {X 0,Y 286.517,Z 681.728,A -85,B 0,C 180,E1 -27502.326,E2 -27502.326} C_VEL
LIN {X 0,Y 277.232,Z 688.935,A -85,B 0,C 180,E1 -27504.472,E2 -27504.472} C_VEL
LIN {X 0,Y 268.625,Z 694.639,A -85,B 0,C 180,E1 -27506.799,E2 -27506.799} C_VEL
LIN {X 0,Y 260.732,Z 698.983,A -85,B 0,C 180,E1 -27509.308,E2 -27509.308} C_VEL
LIN {X 0,Y 253.652,Z 702.054,A -85,B 0,C 180,E1 -27512.002,E2 -27512.002} C_VEL
LIN {X 0,Y 247.324,Z 703.941,A -85,B 0,C 180,E1 -27514.862,E2 -27514.862} C_VEL
LIN {X 0,Y 241.995,Z 704.665,A -85,B 0,C 180,E1 -27517.897,E2 -27517.897} C_VEL
LIN {X 0,Y 237.642,Z 704.25,A -85,B 0,C 180,E1 -27521.082,E2 -27521.082} C_VEL
LIN {X 0,Y 234.059,Z 702.682,A -85,B 0,C 180,E1 -27524.376,E2 -27524.376} C_VEL
LIN {X 0,Y 231.719,Z 699.976,A -85,B 0,C 180,E1 -27527.784,E2 -27527.784} C_VEL
LIN {X 0,Y 230.39,Z 696.06,A -85,B 0,C 180,E1 -27531.257,E2 -27531.257} C_VEL
LIN {X 0,Y 229.967,Z 690.82,A -85,B 0,C 180,E1 -27534.758,E2 -27534.758} C_VEL
LIN {X 0,Y 230.237,Z 684.066,A -85,B 0,C 180,E1 -27538.257,E2 -27538.257} C_VEL
LIN {X 0,Y 230.489,Z 677.744,A -85,B 0,C 180,E1 -27540.871,E2 -27540.871} C_VEL
LIN {X 0,Y 230.748,Z 670.083,A -85,B 0,C 180,E1 -27543.481,E2 -27543.481} C_VEL
LIN {X 0,Y 230.901,Z 662.511,A -85,B 0,C 180,E1 -27545.658,E2 -27545.658} C_VEL
LIN {X 0,Y 231.347,Z 651.682,A -85,B 0,C 180,E1 -27548.269,E2 -27548.269} C_VEL
LIN {X 0,Y 231.943,Z 638.429,A -85,B 0,C 180,E1 -27550.88,E2 -27550.88} C_VEL
LIN {X 0,Y 232.542,Z 626.322,A -85,B 0,C 180,E1 -27552.836,E2 -27552.836} C_VEL
LIN {X 0,Y 233.298,Z 613.297,A -85,B 0,C 180,E1 -27554.564,E2 -27554.564} C_VEL
LIN {X 0,Y 234.079,Z 598.928,A -85,B 0,C 180,E1 -27556.086,E2 -27556.086} C_VEL
LIN {X 0,Y 234.716,Z 583.865,A -85,B 0,C 180,E1 -27557.316,E2 -27557.316} C_VEL
LIN {X 0,Y 235.736,Z 554.769,A -85,B 0,C 180,E1 -27559.022,E2 -27559.022} C_VEL
LIN {X 0,Y 238.563,Z 480.389,A -85,B 0,C 180,E1 -27563.117,E2 -27563.117} C_VEL
LIN {X 0,Y 236.525,Z 450.754,A -85,B 0,C 180,E1 -27564.728,E2 -27564.728} C_VEL
LIN {X 0,Y 236.382,Z 439.685,A -85,B 0,C 180,E1 -27565.329,E2 -27565.329} C_VEL
LIN {X 0,Y 239.396,Z 414.35,A -85,B 0,C 180,E1 -27570.313,E2 -27570.313} C_VEL
LIN {X 0,Y 240.214,Z 406.294,A -85,B 0,C 180,E1 -27571.894,E2 -27571.894} C_VEL
LIN {X 0,Y 235.448,Z 384.391,A -85,B 0,C 180,E1 -27576.56,E2 -27576.56} C_VEL
LIN {X 0,Y 232.075,Z 369.127,A -85,B 0,C 180,E1 -27579.953,E2 -27579.953} C_VEL
LIN {X 0,Y 232.036,Z 369.138,A -85,B 0,C 180,E1 -27583.972,E2 -27583.972} C_VEL
LIN {X 0,Y 232.007,Z 369.141,A -85,B 0,C 180,E1 -27588.38,E2 -27588.38} C_VEL
LIN {X 0,Y 232.002,Z 369.136,A -85,B 0,C 180,E1 -27592.856,E2 -27592.856} C_VEL
LIN {X 0,Y 232.031,Z 369.138,A -85,B 0,C 180,E1 -27595.385,E2 -27595.385} C_VEL
LIN {X 0,Y 233.058,Z 372.01,A -85,B 0,C 180,E1 -27595.695,E2 -27595.695} C_VEL
LIN {X 0,Y 234.642,Z 374.173,A -85,B 0,C 180,E1 -27596.077,E2 -27596.077} C_VEL
LIN {X 0,Y 243.654,Z 389.356,A -85,B 0,C 180,E1 -27598.221,E2 -27598.221} C_VEL
LIN {X 0,Y 251.857,Z 404.95,A -85,B 0,C 180,E1 -27600.055,E2 -27600.055} C_VEL
LIN {X 0,Y 257.322,Z 417.071,A -85,B 0,C 180,E1 -27601.249,E2 -27601.249} C_VEL
LIN {X 0,Y 255.39,Z 468.57,A -85,B 0,C 180,E1 -27602.644,E2 -27602.644} C_VEL
LIN {X 0,Y 254.8,Z 488.32,A -85,B 0,C 180,E1 -27603.29,E2 -27603.29} C_VEL
LIN {X 0,Y 253.853,Z 502.782,A -85,B 0,C 180,E1 -27604.077,E2 -27604.077} C_VEL
LIN {X 0,Y 252.385,Z 515.914,A -85,B 0,C 180,E1 -27605.071,E2 -27605.071} C_VEL
LIN {X 0,Y 250.569,Z 528.327,A -85,B 0,C 180,E1 -27606.307,E2 -27606.307} C_VEL
LIN {X 0,Y 248.53,Z 540.452,A -85,B 0,C 180,E1 -27607.855,E2 -27607.855} C_VEL
LIN {X 0,Y 246.28,Z 551.573,A -85,B 0,C 180,E1 -27609.611,E2 -27609.611} C_VEL
LIN {X 0,Y 243.774,Z 561.839,A -85,B 0,C 180,E1 -27611.575,E2 -27611.575} C_VEL
LIN {X 0,Y 241.069,Z 572.056,A -85,B 0,C 180,E1 -27613.977,E2 -27613.977} C_VEL
LIN {X 0,Y 238.69,Z 580.491,A -85,B 0,C 180,E1 -27616.423,E2 -27616.423} C_VEL
LIN {X 0,Y 236.376,Z 588.574,A -85,B 0,C 180,E1 -27619.327,E2 -27619.327} C_VEL
LIN {X 0,Y 234.455,Z 595.09,A -85,B 0,C 180,E1 -27622.274,E2 -27622.274} C_VEL
LIN {X 0,Y 232.952,Z 600.867,A -85,B 0,C 180,E1 -27625.689,E2 -27625.689} C_VEL
LIN {X 0,Y 232.013,Z 604.243,A -85,B 0,C 180,E1 -27628.27,E2 -27628.27} C_VEL
LIN {X 0,Y 231.45,Z 607.435,A -85,B 0,C 180,E1 -27631.735,E2 -27631.735} C_VEL
LIN {X 0,Y 231.485,Z 609.278,A -85,B 0,C 180,E1 -27635.209,E2 -27635.209} C_VEL
LIN {X 0,Y 231.878,Z 609.85,A -85,B 0,C 180,E1 -27638.687,E2 -27638.687} C_VEL
LIN {X 0,Y 232.835,Z 609.129,A -85,B 0,C 180,E1 -27642.157,E2 -27642.157} C_VEL
LIN {X 0,Y 234.485,Z 607.084,A -85,B 0,C 180,E1 -27645.596,E2 -27645.596} C_VEL
LIN {X 0,Y 236.76,Z 603.658,A -85,B 0,C 180,E1 -27648.992,E2 -27648.992} C_VEL
LIN {X 0,Y 239.619,Z 598.746,A -85,B 0,C 180,E1 -27652.335,E2 -27652.335} C_VEL
LIN {X 0,Y 242.177,Z 593.96,A -85,B 0,C 180,E1 -27654.796,E2 -27654.796} C_VEL
LIN {X 0,Y 245.128,Z 588.141,A -85,B 0,C 180,E1 -27657.207,E2 -27657.207} C_VEL
LIN {X 0,Y 248.296,Z 581.124,A -85,B 0,C 180,E1 -27659.583,E2 -27659.583} C_VEL
LIN {X 0,Y 251.88,Z 572.635,A -85,B 0,C 180,E1 -27661.895,E2 -27661.895} C_VEL
LIN {X 0,Y 255.772,Z 562.307,A -85,B 0,C 180,E1 -27664.153,E2 -27664.153} C_VEL
LIN {X 0,Y 258.66,Z 553.457,A -85,B 0,C 180,E1 -27665.761,E2 -27665.761} C_VEL
LIN {X 0,Y 262.03,Z 541.894,A -85,B 0,C 180,E1 -27667.456,E2 -27667.456} C_VEL
LIN {X 0,Y 265.043,Z 529.675,A -85,B 0,C 180,E1 -27668.878,E2 -27668.878} C_VEL
LIN {X 0,Y 267.277,Z 517.203,A -85,B 0,C 180,E1 -27670.062,E2 -27670.062} C_VEL
LIN {X 0,Y 269.177,Z 503.299,A -85,B 0,C 180,E1 -27671.053,E2 -27671.053} C_VEL
LIN {X 0,Y 270.422,Z 489.443,A -85,B 0,C 180,E1 -27671.753,E2 -27671.753} C_VEL
LIN {X 0,Y 271.23,Z 471.25,A -85,B 0,C 180,E1 -27672.325,E2 -27672.325} C_VEL
LIN {X 0,Y 272.978,Z 434.31,A -85,B 0,C 180,E1 -27673.27,E2 -27673.27} C_VEL
LIN {X 0,Y 266.399,Z 421.322,A -85,B 0,C 180,E1 -27674.992,E2 -27674.992} C_VEL
LIN {X 0,Y 257.903,Z 406.626,A -85,B 0,C 180,E1 -27677.348,E2 -27677.348} C_VEL
LIN {X 0,Y 250.308,Z 394.98,A -85,B 0,C 180,E1 -27679.624,E2 -27679.624} C_VEL
LIN {X 0,Y 244.591,Z 386.918,A -85,B 0,C 180,E1 -27681.472,E2 -27681.472} C_VEL
LIN {X 0,Y 242.162,Z 383.481,A -85,B 0,C 180,E1 -27682.306,E2 -27682.306} C_VEL
LIN {X 0,Y 239.49,Z 379.725,A -85,B 0,C 180,E1 -27683.261,E2 -27683.261} C_VEL
LIN {X 0,Y 236.454,Z 376.015,A -85,B 0,C 180,E1 -27684.371,E2 -27684.371} C_VEL
LIN {X 0,Y 235.43,Z 374.335,A -85,B 0,C 180,E1 -27684.78,E2 -27684.78} C_VEL
LIN {X 0,Y 233.126,Z 372.139,A -85,B 0,C 180,E1 -27685.646,E2 -27685.646} C_VEL
LIN {X 0,Y 232.098,Z 369.578,A -85,B 0,C 180,E1 -27686.126,E2 -27686.126} C_VEL
LIN {X 0,Y 232.03,Z 369.116,A -85,B 0,C 180,E1 -27686.179,E2 -27686.179} C_VEL
LIN {X 0,Y 232.032,Z 369.133,A -85,B 0,C 180,E1 -27691.118,E2 -27691.118} C_VEL
LIN {X 0,Y 232.221,Z 369.152,A -85,B 0,C 180,E1 -27695.683,E2 -27695.683} C_VEL
LIN {X 0,Y 236.073,Z 387.034,A -85,B 0,C 180,E1 -27696.674,E2 -27696.674} C_VEL
LIN {X 0,Y 237.571,Z 393.418,A -85,B 0,C 180,E1 -27697.021,E2 -27697.021} C_VEL
LIN {X 0,Y 235.361,Z 466.034,A -85,B 0,C 180,E1 -27700.891,E2 -27700.891} C_VEL
LIN {X 0,Y 234.74,Z 487.601,A -85,B 0,C 180,E1 -27702.134,E2 -27702.134} C_VEL
LIN {X 0,Y 234.177,Z 501.942,A -85,B 0,C 180,E1 -27703.251,E2 -27703.251} C_VEL
LIN {X 0,Y 233.52,Z 515.111,A -85,B 0,C 180,E1 -27704.561,E2 -27704.561} C_VEL
LIN {X 0,Y 232.703,Z 530.648,A -85,B 0,C 180,E1 -27706.509,E2 -27706.509} C_VEL
LIN {X 0,Y 232.026,Z 543.299,A -85,B 0,C 180,E1 -27708.463,E2 -27708.463} C_VEL
LIN {X 0,Y 231.386,Z 555.029,A -85,B 0,C 180,E1 -27710.635,E2 -27710.635} C_VEL
LIN {X 0,Y 230.894,Z 565.908,A -85,B 0,C 180,E1 -27713.03,E2 -27713.03} C_VEL
LIN {X 0,Y 230.664,Z 575.914,A -85,B 0,C 180,E1 -27715.646,E2 -27715.646} C_VEL
LIN {X 0,Y 230.775,Z 585.707,A -85,B 0,C 180,E1 -27718.695,E2 -27718.695} C_VEL
LIN {X 0,Y 231.124,Z 593.845,A -85,B 0,C 180,E1 -27721.736,E2 -27721.736} C_VEL
LIN {X 0,Y 231.953,Z 599.667,A -85,B 0,C 180,E1 -27724.329,E2 -27724.329} C_VEL
LIN {X 0,Y 233.844,Z 606.077,A -85,B 0,C 180,E1 -27727.746,E2 -27727.746} C_VEL
LIN {X 0,Y 236.398,Z 611.045,A -85,B 0,C 180,E1 -27731.104,E2 -27731.104} C_VEL
LIN {X 0,Y 238.854,Z 613.83,A -85,B 0,C 180,E1 -27733.568,E2 -27733.568} C_VEL
LIN {X 0,Y 243.101,Z 616.473,A -85,B 0,C 180,E1 -27736.746,E2 -27736.746} C_VEL
LIN {X 0,Y 248.399,Z 617.798,A -85,B 0,C 180,E1 -27739.778,E2 -27739.778} C_VEL
LIN {X 0,Y 254.295,Z 617.86,A -85,B 0,C 180,E1 -27742.682,E2 -27742.682} C_VEL
LIN {X 0,Y 260.836,Z 616.674,A -85,B 0,C 180,E1 -27745.446,E2 -27745.446} C_VEL
LIN {X 0,Y 265.144,Z 615.29,A -85,B 0,C 180,E1 -27747.059,E2 -27747.059} C_VEL
LIN {X 0,Y 267.698,Z 614.293,A -85,B 0,C 180,E1 -27748.185,E2 -27748.185} C_VEL
LIN {X 0,Y 273.23,Z 611.522,A -85,B 0,C 180,E1 -27751.728,E2 -27751.728} C_VEL
LIN {X 0,Y 275.81,Z 609.964,A -85,B 0,C 180,E1 -27752.783,E2 -27752.783} C_VEL
LIN {X 0,Y 276.873,Z 609.307,A -85,B 0,C 180,E1 -27753.096,E2 -27753.096} C_VEL
LIN {X 0,Y 285.429,Z 603.63,A -85,B 0,C 180,E1 -27755.218,E2 -27755.218} C_VEL
LIN {X 0,Y 294.953,Z 596.074,A -85,B 0,C 180,E1 -27757.269,E2 -27757.269} C_VEL
LIN {X 0,Y 303.652,Z 587.844,A -85,B 0,C 180,E1 -27758.946,E2 -27758.946} C_VEL
LIN {X 0,Y 312.603,Z 577.926,A -85,B 0,C 180,E1 -27760.526,E2 -27760.526} C_VEL
LIN {X 0,Y 320.469,Z 567.73,A -85,B 0,C 180,E1 -27761.808,E2 -27761.808} C_VEL
LIN {X 0,Y 328.466,Z 555.666,A -85,B 0,C 180,E1 -27763.031,E2 -27763.031} C_VEL
LIN {X 0,Y 326.828,Z 558.48,A -85,B 0,C 180,E1 -27763.224,E2 -27763.224} C_VEL
LIN {X 0,Y 318.057,Z 572.444,A -85,B 0,C 180,E1 -27764.07,E2 -27764.07} C_VEL
LIN {X 0,Y 309.609,Z 584.131,A -85,B 0,C 180,E1 -27765.009,E2 -27765.009} C_VEL
LIN {X 0,Y 299.268,Z 596.617,A -85,B 0,C 180,E1 -27766.333,E2 -27766.333} C_VEL
LIN {X 0,Y 289.418,Z 607.077,A -85,B 0,C 180,E1 -27767.809,E2 -27767.809} C_VEL
LIN {X 0,Y 280.101,Z 615.931,A -85,B 0,C 180,E1 -27769.444,E2 -27769.444} C_VEL
LIN {X 0,Y 272.514,Z 622.372,A -85,B 0,C 180,E1 -27770.97,E2 -27770.97} C_VEL
LIN {X 0,Y 263.199,Z 629.607,A -85,B 0,C 180,E1 -27773.217,E2 -27773.217} C_VEL
LIN {X 0,Y 254.67,Z 635.441,A -85,B 0,C 180,E1 -27775.678,E2 -27775.678} C_VEL
LIN {X 0,Y 248.881,Z 639.037,A -85,B 0,C 180,E1 -27777.674,E2 -27777.674} C_VEL
LIN {X 0,Y 241.994,Z 642.752,A -85,B 0,C 180,E1 -27780.524,E2 -27780.524} C_VEL
LIN {X 0,Y 236.049,Z 645.364,A -85,B 0,C 180,E1 -27783.569,E2 -27783.569} C_VEL
LIN {X 0,Y 231.309,Z 646.932,A -85,B 0,C 180,E1 -27786.817,E2 -27786.817} C_VEL
LIN {X 0,Y 227.88,Z 647.512,A -85,B 0,C 180,E1 -27790.238,E2 -27790.238} C_VEL
LIN {X 0,Y 226.486,Z 647.427,A -85,B 0,C 180,E1 -27792.217,E2 -27792.217} C_VEL
LIN {X 0,Y 224.036,Z 652.737,A -85,B 0,C 180,E1 -27795.991,E2 -27795.991} C_VEL
LIN {X 0,Y 223.303,Z 655.853,A -85,B 0,C 180,E1 -27799.152,E2 -27799.152} C_VEL
LIN {X 0,Y 223.757,Z 658.233,A -85,B 0,C 180,E1 -27802.806,E2 -27802.806} C_VEL
LIN {X 0,Y 224.163,Z 658.736,A -85,B 0,C 180,E1 -27803.89,E2 -27803.89} C_VEL
LIN {X 0,Y 224.057,Z 667.984,A -85,B 0,C 180,E1 -27806.415,E2 -27806.415} C_VEL
LIN {X 0,Y 223.867,Z 676.084,A -85,B 0,C 180,E1 -27809.103,E2 -27809.103} C_VEL
LIN {X 0,Y 223.595,Z 682.76,A -85,B 0,C 180,E1 -27811.795,E2 -27811.795} C_VEL
LIN {X 0,Y 223.323,Z 688.244,A -85,B 0,C 180,E1 -27814.497,E2 -27814.497} C_VEL
LIN {X 0,Y 223.37,Z 694.134,A -85,B 0,C 180,E1 -27818.112,E2 -27818.112} C_VEL
LIN {X 0,Y 223.901,Z 697.665,A -85,B 0,C 180,E1 -27820.818,E2 -27820.818} C_VEL
LIN {X 0,Y 225.816,Z 701.28,A -85,B 0,C 180,E1 -27824.368,E2 -27824.368} C_VEL
LIN {X 0,Y 228.834,Z 703.713,A -85,B 0,C 180,E1 -27827.824,E2 -27827.824} C_VEL
LIN {X 0,Y 232.837,Z 705.006,A -85,B 0,C 180,E1 -27831.161,E2 -27831.161} C_VEL
LIN {X 0,Y 237.674,Z 705.18,A -85,B 0,C 180,E1 -27834.368,E2 -27834.368} C_VEL
LIN {X 0,Y 243.669,Z 704.238,A -85,B 0,C 180,E1 -27837.383,E2 -27837.383} C_VEL
LIN {X 0,Y 250.664,Z 702.138,A -85,B 0,C 180,E1 -27840.197,E2 -27840.197} C_VEL
LIN {X 0,Y 258.875,Z 698.617,A -85,B 0,C 180,E1 -27842.99,E2 -27842.99} C_VEL
LIN {X 0,Y 266.829,Z 694.333,A -85,B 0,C 180,E1 -27845.276,E2 -27845.276} C_VEL
LIN {X 0,Y 276.031,Z 688.427,A -85,B 0,C 180,E1 -27847.518,E2 -27847.518} C_VEL
LIN {X 0,Y 285.865,Z 681.023,A -85,B 0,C 180,E1 -27849.573,E2 -27849.573} C_VEL
LIN {X 0,Y 296.271,Z 671.929,A -85,B 0,C 180,E1 -27851.451,E2 -27851.451} C_VEL
LIN {X 0,Y 305.991,Z 662.076,A -85,B 0,C 180,E1 -27852.968,E2 -27852.968} C_VEL
LIN {X 0,Y 315.053,Z 651.569,A -85,B 0,C 180,E1 -27854.203,E2 -27854.203} C_VEL
LIN {X 0,Y 320.243,Z 644.867,A -85,B 0,C 180,E1 -27854.854,E2 -27854.854} C_VEL
LIN {X 0,Y 318.929,Z 646.611,A -85,B 0,C 180,E1 -27855.348,E2 -27855.348} C_VEL
LIN {X 0,Y 309.34,Z 658.35,A -85,B 0,C 180,E1 -27856.622,E2 -27856.622} C_VEL
LIN {X 0,Y 300.586,Z 667.661,A -85,B 0,C 180,E1 -27857.937,E2 -27857.937} C_VEL
LIN {X 0,Y 291.26,Z 676.366,A -85,B 0,C 180,E1 -27859.51,E2 -27859.51} C_VEL
LIN {X 0,Y 283.636,Z 682.681,A -85,B 0,C 180,E1 -27860.97,E2 -27860.97} C_VEL
LIN {X 0,Y 273.99,Z 689.665,A -85,B 0,C 180,E1 -27863.075,E2 -27863.075} C_VEL
LIN {X 0,Y 265.004,Z 695.169,A -85,B 0,C 180,E1 -27865.37,E2 -27865.37} C_VEL
LIN {X 0,Y 258.694,Z 698.411,A -85,B 0,C 180,E1 -27867.213,E2 -27867.213} C_VEL
LIN {X 0,Y 251,Z 701.654,A -85,B 0,C 180,E1 -27869.847,E2 -27869.847} C_VEL
LIN {X 0,Y 244.113,Z 703.718,A -85,B 0,C 180,E1 -27872.672,E2 -27872.672} C_VEL
LIN {X 0,Y 238.019,Z 704.644,A -85,B 0,C 180,E1 -27875.67,E2 -27875.67} C_VEL
LIN {X 0,Y 233.098,Z 704.445,A -85,B 0,C 180,E1 -27878.864,E2 -27878.864} C_VEL
LIN {X 0,Y 229.011,Z 703.123,A -85,B 0,C 180,E1 -27882.191,E2 -27882.191} C_VEL
LIN {X 0,Y 225.985,Z 700.67,A -85,B 0,C 180,E1 -27885.643,E2 -27885.643} C_VEL
LIN {X 0,Y 223.958,Z 697.021,A -85,B 0,C 180,E1 -27889.185,E2 -27889.185} C_VEL
LIN {X 0,Y 223.259,Z 692.17,A -85,B 0,C 180,E1 -27892.791,E2 -27892.791} C_VEL
LIN {X 0,Y 223.189,Z 685.844,A -85,B 0,C 180,E1 -27896.402,E2 -27896.402} C_VEL
LIN {X 0,Y 223.581,Z 678.934,A -85,B 0,C 180,E1 -27899.552,E2 -27899.552} C_VEL
LIN {X 0,Y 223.859,Z 671.642,A -85,B 0,C 180,E1 -27902.242,E2 -27902.242} C_VEL
LIN {X 0,Y 223.999,Z 662.78,A -85,B 0,C 180,E1 -27904.934,E2 -27904.934} C_VEL
LIN {X 0,Y 224.438,Z 651.075,A -85,B 0,C 180,E1 -27907.848,E2 -27907.848} C_VEL
LIN {X 0,Y 224.978,Z 637.819,A -85,B 0,C 180,E1 -27910.54,E2 -27910.54} C_VEL
LIN {X 0,Y 225.571,Z 625.596,A -85,B 0,C 180,E1 -27912.555,E2 -27912.555} C_VEL
LIN {X 0,Y 226.411,Z 610.631,A -85,B 0,C 180,E1 -27914.559,E2 -27914.559} C_VEL
LIN {X 0,Y 227.19,Z 595.904,A -85,B 0,C 180,E1 -27916.11,E2 -27916.11} C_VEL
LIN {X 0,Y 227.789,Z 579.44,A -85,B 0,C 180,E1 -27917.403,E2 -27917.403} C_VEL
LIN {X 0,Y 230.598,Z 502.265,A -85,B 0,C 180,E1 -27921.904,E2 -27921.904} C_VEL
LIN {X 0,Y 231.375,Z 479.848,A -85,B 0,C 180,E1 -27923.176,E2 -27923.176} C_VEL
LIN {X 0,Y 229.427,Z 450.515,A -85,B 0,C 180,E1 -27924.82,E2 -27924.82} C_VEL
LIN {X 0,Y 229.307,Z 439.642,A -85,B 0,C 180,E1 -27925.44,E2 -27925.44} C_VEL
LIN {X 0,Y 232.384,Z 414.219,A -85,B 0,C 180,E1 -27930.574,E2 -27930.574} C_VEL
LIN {X 0,Y 233.171,Z 407.313,A -85,B 0,C 180,E1 -27931.961,E2 -27931.961} C_VEL
LIN {X 0,Y 228.498,Z 385.851,A -85,B 0,C 180,E1 -27936.624,E2 -27936.624} C_VEL
LIN {X 0,Y 225.032,Z 370.002,A -85,B 0,C 180,E1 -27940.206,E2 -27940.206} C_VEL
LIN {X 0,Y 224.997,Z 370.013,A -85,B 0,C 180,E1 -27944.273,E2 -27944.273} C_VEL
LIN {X 0,Y 224.972,Z 370.01,A -85,B 0,C 180,E1 -27949.169,E2 -27949.169} C_VEL
LIN {X 0,Y 224.949,Z 370.021,A -85,B 0,C 180,E1 -27953.996,E2 -27953.996} C_VEL
LIN {X 0,Y 225.988,Z 372.909,A -85,B 0,C 180,E1 -27954.329,E2 -27954.329} C_VEL
LIN {X 0,Y 227.796,Z 375.291,A -85,B 0,C 180,E1 -27954.792,E2 -27954.792} C_VEL
LIN {X 0,Y 237.252,Z 390.889,A -85,B 0,C 180,E1 -27957.175,E2 -27957.175} C_VEL
LIN {X 0,Y 245.453,Z 406.38,A -85,B 0,C 180,E1 -27959.111,E2 -27959.111} C_VEL
LIN {X 0,Y 251.287,Z 419.197,A -85,B 0,C 180,E1 -27960.447,E2 -27960.447} C_VEL
LIN {X 0,Y 249.356,Z 467.788,A -85,B 0,C 180,E1 -27961.785,E2 -27961.785} C_VEL
LIN {X 0,Y 248.713,Z 488.493,A -85,B 0,C 180,E1 -27962.464,E2 -27962.464} C_VEL
LIN {X 0,Y 247.704,Z 503.215,A -85,B 0,C 180,E1 -27963.27,E2 -27963.27} C_VEL
LIN {X 0,Y 246.206,Z 516.426,A -85,B 0,C 180,E1 -27964.288,E2 -27964.288} C_VEL
LIN {X 0,Y 244.149,Z 529.768,A -85,B 0,C 180,E1 -27965.644,E2 -27965.644} C_VEL
LIN {X 0,Y 242.055,Z 541.759,A -85,B 0,C 180,E1 -27967.23,E2 -27967.23} C_VEL
LIN {X 0,Y 239.715,Z 552.786,A -85,B 0,C 180,E1 -27969.026,E2 -27969.026} C_VEL
LIN {X 0,Y 236.796,Z 564.155,A -85,B 0,C 180,E1 -27971.293,E2 -27971.293} C_VEL
LIN {X 0,Y 233.866,Z 574.603,A -85,B 0,C 180,E1 -27973.916,E2 -27973.916} C_VEL
LIN {X 0,Y 231.158,Z 583.943,A -85,B 0,C 180,E1 -27976.864,E2 -27976.864} C_VEL
LIN {X 0,Y 229.177,Z 590.52,A -85,B 0,C 180,E1 -27979.434,E2 -27979.434} C_VEL
LIN {X 0,Y 227.492,Z 596.008,A -85,B 0,C 180,E1 -27982.036,E2 -27982.036} C_VEL
LIN {X 0,Y 225.923,Z 601.752,A -85,B 0,C 180,E1 -27985.555,E2 -27985.555} C_VEL
LIN {X 0,Y 224.953,Z 605.106,A -85,B 0,C 180,E1 -27988.216,E2 -27988.216} C_VEL
LIN {X 0,Y 224.389,Z 608.256,A -85,B 0,C 180,E1 -27991.789,E2 -27991.789} C_VEL
LIN {X 0,Y 224.43,Z 610.07,A -85,B 0,C 180,E1 -27995.373,E2 -27995.373} C_VEL
LIN {X 0,Y 224.88,Z 610.611,A -85,B 0,C 180,E1 -27998.96,E2 -27998.96} C_VEL
LIN {X 0,Y 225.903,Z 609.862,A -85,B 0,C 180,E1 -28002.536,E2 -28002.536} C_VEL
LIN {X 0,Y 227.663,Z 607.784,A -85,B 0,C 180,E1 -28006.076,E2 -28006.076} C_VEL
LIN {X 0,Y 230.043,Z 604.328,A -85,B 0,C 180,E1 -28009.569,E2 -28009.569} C_VEL
LIN {X 0,Y 233.056,Z 599.38,A -85,B 0,C 180,E1 -28012.999,E2 -28012.999} C_VEL
LIN {X 0,Y 235.731,Z 594.559,A -85,B 0,C 180,E1 -28015.522,E2 -28015.522} C_VEL
LIN {X 0,Y 239.33,Z 587.543,A -85,B 0,C 180,E1 -28018.426,E2 -28018.426} C_VEL
LIN {X 0,Y 243.347,Z 578.966,A -85,B 0,C 180,E1 -28021.206,E2 -28021.206} C_VEL
LIN {X 0,Y 247.24,Z 569.875,A -85,B 0,C 180,E1 -28023.535,E2 -28023.535} C_VEL
LIN {X 0,Y 250.895,Z 559.807,A -85,B 0,C 180,E1 -28025.647,E2 -28025.647} C_VEL
LIN {X 0,Y 254.516,Z 548.668,A -85,B 0,C 180,E1 -28027.51,E2 -28027.51} C_VEL
LIN {X 0,Y 258.015,Z 536.292,A -85,B 0,C 180,E1 -28029.138,E2 -28029.138} C_VEL
LIN {X 0,Y 260.53,Z 524.445,A -85,B 0,C 180,E1 -28030.42,E2 -28030.42} C_VEL
LIN {X 0,Y 262.735,Z 511.269,A -85,B 0,C 180,E1 -28031.523,E2 -28031.523} C_VEL
LIN {X 0,Y 264.37,Z 497.477,A -85,B 0,C 180,E1 -28032.377,E2 -28032.377} C_VEL
LIN {X 0,Y 265.353,Z 483.755,A -85,B 0,C 180,E1 -28032.952,E2 -28032.952} C_VEL
LIN {X 0,Y 267.354,Z 442.422,A -85,B 0,C 180,E1 -28034.049,E2 -28034.049} C_VEL
LIN {X 0,Y 267.603,Z 436.832,A -85,B 0,C 180,E1 -28034.199,E2 -28034.199} C_VEL
LIN {X 0,Y 260.824,Z 423.545,A -85,B 0,C 180,E1 -28036.062,E2 -28036.062} C_VEL
LIN {X 0,Y 253.107,Z 410.237,A -85,B 0,C 180,E1 -28038.314,E2 -28038.314} C_VEL
LIN {X 0,Y 244.98,Z 397.683,A -85,B 0,C 180,E1 -28040.892,E2 -28040.892} C_VEL
LIN {X 0,Y 238.503,Z 388.631,A -85,B 0,C 180,E1 -28043.137,E2 -28043.137} C_VEL
LIN {X 0,Y 235.422,Z 384.468,A -85,B 0,C 180,E1 -28044.283,E2 -28044.283} C_VEL
LIN {X 0,Y 232.185,Z 380.142,A -85,B 0,C 180,E1 -28045.552,E2 -28045.552} C_VEL
LIN {X 0,Y 229.778,Z 377.305,A -85,B 0,C 180,E1 -28046.525,E2 -28046.525} C_VEL
LIN {X 0,Y 228.898,Z 375.503,A -85,B 0,C 180,E1 -28046.933,E2 -28046.933} C_VEL
LIN {X 0,Y 226.443,Z 373.537,A -85,B 0,C 180,E1 -28047.94,E2 -28047.94} C_VEL
LIN {X 0,Y 225.218,Z 371.174,A -85,B 0,C 180,E1 -28048.539,E2 -28048.539} C_VEL
LIN {X 0,Y 224.958,Z 370.004,A -85,B 0,C 180,E1 -28048.727,E2 -28048.727} C_VEL
LIN {X 0,Y 224.987,Z 370.015,A -85,B 0,C 180,E1 -28052.16,E2 -28052.16} C_VEL
LIN {X 0,Y 225.181,Z 369.984,A -85,B 0,C 180,E1 -28055.638,E2 -28055.638} C_VEL
LIN {X 0,Y 228.882,Z 387.496,A -85,B 0,C 180,E1 -28056.649,E2 -28056.649} C_VEL
LIN {X 0,Y 230.429,Z 394.507,A -85,B 0,C 180,E1 -28057.042,E2 -28057.042} C_VEL
LIN {X 0,Y 228.179,Z 471.22,A -85,B 0,C 180,E1 -28061.312,E2 -28061.312} C_VEL
LIN {X 0,Y 227.573,Z 490.211,A -85,B 0,C 180,E1 -28062.481,E2 -28062.481} C_VEL
LIN {X 0,Y 226.981,Z 504.738,A -85,B 0,C 180,E1 -28063.695,E2 -28063.695} C_VEL
LIN {X 0,Y 226.153,Z 520.502,A -85,B 0,C 180,E1 -28065.424,E2 -28065.424} C_VEL
LIN {X 0,Y 225.429,Z 535.091,A -85,B 0,C 180,E1 -28067.437,E2 -28067.437} C_VEL
LIN {X 0,Y 224.723,Z 548.29,A -85,B 0,C 180,E1 -28069.675,E2 -28069.675} C_VEL
LIN {X 0,Y 224.057,Z 561.307,A -85,B 0,C 180,E1 -28072.364,E2 -28072.364} C_VEL
LIN {X 0,Y 223.718,Z 572.123,A -85,B 0,C 180,E1 -28075.06,E2 -28075.06} C_VEL
LIN {X 0,Y 223.744,Z 582.734,A -85,B 0,C 180,E1 -28078.206,E2 -28078.206} C_VEL
LIN {X 0,Y 224.02,Z 591.491,A -85,B 0,C 180,E1 -28081.343,E2 -28081.343} C_VEL
LIN {X 0,Y 224.925,Z 598.772,A -85,B 0,C 180,E1 -28084.465,E2 -28084.465} C_VEL
LIN {X 0,Y 226.834,Z 605.584,A -85,B 0,C 180,E1 -28087.987,E2 -28087.987} C_VEL
LIN {X 0,Y 229.451,Z 610.871,A -85,B 0,C 180,E1 -28091.444,E2 -28091.444} C_VEL
LIN {X 0,Y 231.986,Z 614.006,A -85,B 0,C 180,E1 -28093.977,E2 -28093.977} C_VEL
LIN {X 0,Y 236.338,Z 617.021,A -85,B 0,C 180,E1 -28097.24,E2 -28097.24} C_VEL
LIN {X 0,Y 241.778,Z 618.739,A -85,B 0,C 180,E1 -28100.343,E2 -28100.343} C_VEL
LIN {X 0,Y 247.883,Z 619.191,A -85,B 0,C 180,E1 -28103.303,E2 -28103.303} C_VEL
LIN {X 0,Y 254.631,Z 618.394,A -85,B 0,C 180,E1 -28106.112,E2 -28106.112} C_VEL
LIN {X 0,Y 262.059,Z 616.334,A -85,B 0,C 180,E1 -28108.758,E2 -28108.758} C_VEL
LIN {X 0,Y 270.078,Z 612.948,A -85,B 0,C 180,E1 -28111.245,E2 -28111.245} C_VEL
LIN {X 0,Y 276.873,Z 609.307,A -85,B 0,C 180,E1 -28113.096,E2 -28113.096} C_VEL
LIN {X 0,Y 279.875,Z 607.438,A -85,B 0,C 180,E1 -28114.072,E2 -28114.072} C_VEL
LIN {X 0,Y 287.146,Z 602.289,A -85,B 0,C 180,E1 -28117.195,E2 -28117.195} C_VEL
LIN {X 0,Y 290.743,Z 599.464,A -85,B 0,C 180,E1 -28118.201,E2 -28118.201} C_VEL
LIN {X 0,Y 291.336,Z 598.971,A -85,B 0,C 180,E1 -28118.322,E2 -28118.322} C_VEL
LIN {X 0,Y 301.409,Z 590.137,A -85,B 0,C 180,E1 -28120.157,E2 -28120.157} C_VEL
LIN {X 0,Y 311.527,Z 579.492,A -85,B 0,C 180,E1 -28121.825,E2 -28121.825} C_VEL
LIN {X 0,Y 316.054,Z 574.083,A -85,B 0,C 180,E1 -28122.527,E2 -28122.527} C_VEL
LIN {X 0,Y 316.715,Z 573.354,A -85,B 0,C 180,E1 -28122.818,E2 -28122.818} C_VEL
LIN {X 0,Y 306.258,Z 586.855,A -85,B 0,C 180,E1 -28123.909,E2 -28123.909} C_VEL
LIN {X 0,Y 297.049,Z 597.259,A -85,B 0,C 180,E1 -28125.024,E2 -28125.024} C_VEL
LIN {X 0,Y 287.076,Z 607.26,A -85,B 0,C 180,E1 -28126.426,E2 -28126.426} C_VEL
LIN {X 0,Y 277.462,Z 615.795,A -85,B 0,C 180,E1 -28128.011,E2 -28128.011} C_VEL
LIN {X 0,Y 267.089,Z 623.958,A -85,B 0,C 180,E1 -28130.02,E2 -28130.02} C_VEL
LIN {X 0,Y 257.577,Z 630.583,A -85,B 0,C 180,E1 -28132.276,E2 -28132.276} C_VEL
LIN {X 0,Y 248.855,Z 635.93,A -85,B 0,C 180,E1 -28134.759,E2 -28134.759} C_VEL
LIN {X 0,Y 242.917,Z 639.14,A -85,B 0,C 180,E1 -28136.779,E2 -28136.779} C_VEL
LIN {X 0,Y 235.841,Z 642.448,A -85,B 0,C 180,E1 -28139.675,E2 -28139.675} C_VEL
LIN {X 0,Y 229.73,Z 644.694,A -85,B 0,C 180,E1 -28142.783,E2 -28142.783} C_VEL
LIN {X 0,Y 224.831,Z 645.937,A -85,B 0,C 180,E1 -28146.108,E2 -28146.108} C_VEL
LIN {X 0,Y 221.275,Z 646.19,A -85,B 0,C 180,E1 -28149.622,E2 -28149.622} C_VEL
LIN {X 0,Y 220.096,Z 646.036,A -85,B 0,C 180,E1 -28151.202,E2 -28151.202} C_VEL
LIN {X 0,Y 217.899,Z 650.362,A -85,B 0,C 180,E1 -28154.143,E2 -28154.143} C_VEL
LIN {X 0,Y 216.625,Z 653.472,A -85,B 0,C 180,E1 -28156.918,E2 -28156.918} C_VEL
LIN {X 0,Y 216.25,Z 656.466,A -85,B 0,C 180,E1 -28160.679,E2 -28160.679} C_VEL
LIN {X 0,Y 217.288,Z 658.266,A -85,B 0,C 180,E1 -28164.45,E2 -28164.45} C_VEL
